(* IEC 61131-3 sources: FishAndCat/plc, 9 files *)

(* ---- 01_DUTs.st ---- *)
(* ============================================================
   01_DUTs.st — 数据类型定义(DUT)
   项目:智储优控 · 立体仓储仓位优化(2026 ABB杯 赛道一)
   目标平台:ABB AC500 V3(CODESYS V3.5 内核),ST 语言
   导入方法:Automation Builder 中 Application 右键 → 添加对象 → DUT,
            每个 TYPE 建一个 DUT,粘贴对应段落(详见 README_PLC.md)
   口径依据:docs/canonical_assumptions.md(A1-A9/B1-B5/C1-C8)
   ============================================================ *)

(* ---------- ST_Good:货物(题面五元组 + 分配结果字段) ---------- *)
TYPE ST_Good :
STRUCT
    Id          : INT;          // 序号(题面属性1)
    Name        : STRING[32];   // 名称(题面属性2)
    Weight      : REAL;         // 重量 kg(题面属性3)
    Freq        : REAL;         // 访问频次(题面属性4)
    Volume      : REAL;         // 体积 m3(题面属性5)
    Priority    : REAL;         // Rank阶段优先级(λ1*频次+λ2*重量+λ3*体积,归一后)
    Assigned    : BOOL;         // 是否已分配
    X           : INT;          // 分配结果:列(0..19,水平)
    Y           : INT;          // 分配结果:层(0..19,垂直,0=底层)
    Score       : REAL;         // 分配时的多目标评分
    PathLength  : REAL;         // 单程曼哈顿路径长度 m(口径C2)
    ExecTime    : REAL;         // 单程切比雪夫行程时间 s(口径C2)
END_STRUCT
END_TYPE

(* ---------- ST_Slot:仓位 ---------- *)
TYPE ST_Slot :
STRUCT
    X           : INT;          // 列 0..19
    Y           : INT;          // 层 0..19(0=底层)
    Occupied    : BOOL;         // 已占用(含预占用)
    PresetOcc   : BOOL;         // 预占用(题面:坐标能被3整除,解读见 FC_IsPresetOccupied)
    CapCoef     : REAL;         // 承重系数 = 1.0 - 0.02*Y(题面给定)
    MaxWeight   : REAL;         // 限重 = CapCoef * BASE_CAP(口径A6)
    MaxVolume   : REAL;         // 容积上限 = CELL_VOL(口径B4)
    GoodsId     : INT;          // 存放的货物Id,0=无
END_STRUCT
END_TYPE

(* ---------- ST_Stats:统计信息(决赛可视化统计栏数据源) ---------- *)
TYPE ST_Stats :
STRUCT
    PlacedCnt      : INT;       // 成功入库件数
    FailedCnt      : INT;       // 无可行位件数(边界:必须可见可报警)
    TotalTime2Way  : REAL;      // 入库总时间 s,双程口径(C1)
    AvgTime        : REAL;      // 平均单件双程时间 s
    ExpRetrieval   : REAL;      // 期望取货时间 s,频次加权单程(C3)
    Energy         : REAL;      // 能耗代理 Σ重量*高度 kg·m(C4)
    CogHeight      : REAL;      // 载荷重心高度 m(C6)
    PathTotal2Way  : REAL;      // 路径总长 m,双程曼哈顿(C5 损耗代理)
    UtilPct        : REAL;      // 空间利用率 =已占/400(C7,含预占)
    ViolCnt        : INT;       // 约束违规数,必须恒为0(C8)
    SwapCnt        : INT;       // 局部搜索接受的改进次数
    LsRounds       : INT;       // 局部搜索实际轮数
END_STRUCT
END_TYPE

(* ---------- E_MainState:主程序状态机 ---------- *)
TYPE E_MainState :
(
    STATE_IDLE       := 0,      // 待机
    STATE_INIT       := 10,     // 初始化仓库(预占用/承重)
    STATE_WAIT_INPUT := 20,     // 等待交互输入货物 / 载入演示批次
    STATE_ASSIGN     := 30,     // 批量分配运行中(分片,跨扫描周期)
    STATE_IMPROVE    := 40,     // 局部搜索改进中(分片,跨扫描周期)
    STATE_STATS      := 50,     // 统计计算
    STATE_DONE       := 60,     // 完成,结果可视化
    STATE_FAULT      := 70      // 故障(输入非法/无可行位等,看 GVL_Visu.StatusText)
);
END_TYPE

(* ---- 07_GVL_Data_generated.st ---- *)
(* ============================================================
   07_GVL_Data_generated.st — 生成文件,勿手改!
   由 sim/export_st_vectors.py 生成(seed=2026,N_DEMO=20,
   评分权重 α=1.0 β=0.6 γ=0.4 δ=0.15 = canonical E 默认)
   导入:TYPE 段建 DUT;GVL_Data 段建 GVL;FC_LoadDemoGoods 建 POU(函数)
   ============================================================ *)

(* ---------- DUT:ST_TestVec ---------- *)
TYPE ST_TestVec :
STRUCT
    W        : REAL;   // 货物重量
    F        : REAL;   // 货物频次
    X        : INT;    // 候选仓位列
    Y        : INT;    // 候选仓位层
    WMax     : REAL;   // 归一分母
    FMax     : REAL;
    ExpScore : REAL;   // Python 期望评分(双精度算出,容差1e-3比对)
    ExpTime  : REAL;   // Python 期望切比雪夫时间(匀速口径)
    ExpTimeAccel : REAL;   // Python 期望时间(L1 梯形加减速口径,T22 比对)
END_STRUCT
END_TYPE

(* ---------- DUT:ST_AwraCell(T25 终局布局向量) ---------- *)
TYPE ST_AwraCell :
STRUCT
    Id : INT;    // 货物序号
    X  : INT;    // 终局列
    Y  : INT;    // 终局层
END_STRUCT
END_TYPE

(* ---------- GVL:GVL_Data ---------- *)
VAR_GLOBAL CONSTANT
    N_DEMO    : INT := 20;
    N_TESTVEC : INT := 10;
    N_AWRA    : INT := 20;   // T25 终局向量件数
    AWRA_PLACED : INT := 20;
    AWRA_FAILED : INT := 0;
    LAM_F : REAL := 0.5;   // Rank λ 频次(单源,ST FC_CalcPriority 应引用)
    LAM_W : REAL := 0.35;   // Rank λ 重量
    LAM_V : REAL := 0.15;   // Rank λ 体积
    MAX_LS_ROUNDS : INT := 5;   // LS 最大轮数(单源,ST nMaxLsRounds 应引用)
END_VAR
VAR_GLOBAL
    aTestVec : ARRAY[1..10] OF ST_TestVec := [
        (W := 13.9, F := 1.83, X := 1, Y := 0, WMax := 80.0, FMax := 9.82, ExpScore := 0.122893, ExpTime := 0.500000, ExpTimeAccel := 2.828427),
        (W := 69.5, F := 1.1, X := 5, Y := 2, WMax := 80.0, FMax := 9.82, ExpScore := 0.222415, ExpTime := 4.000000, ExpTimeAccel := 6.324555),
        (W := 50.1, F := 2.02, X := 10, Y := 5, WMax := 80.0, FMax := 9.82, ExpScore := 0.306726, ExpTime := 10.000000, ExpTimeAccel := 11.666667),
        (W := 46.1, F := 3.1, X := 19, Y := 19, WMax := 80.0, FMax := 9.82, ExpScore := 0.891932, ExpTime := 38.000000, ExpTimeAccel := 39.666667),
        (W := 61.3, F := 2.14, X := 0, Y := 1, WMax := 80.0, FMax := 9.82, ExpScore := 0.162936, ExpTime := 2.000000, ExpTimeAccel := 3.666667),
        (W := 51.1, F := 1.11, X := 3, Y := 3, WMax := 80.0, FMax := 9.82, ExpScore := 0.230741, ExpTime := 6.000000, ExpTimeAccel := 7.666667),
        (W := 38.7, F := 4.28, X := 7, Y := 10, WMax := 80.0, FMax := 9.82, ExpScore := 0.524082, ExpTime := 20.000000, ExpTimeAccel := 21.666667),
        (W := 56.0, F := 1.23, X := 15, Y := 1, WMax := 80.0, FMax := 9.82, ExpScore := 0.166878, ExpTime := 7.500000, ExpTimeAccel := 11.500000),
        (W := 78.5, F := 9.82, X := 2, Y := 18, WMax := 80.0, FMax := 9.82, ExpScore := 1.876974, ExpTime := 36.000000, ExpTimeAccel := 37.666667),
        (W := 80.0, F := 1.86, X := 12, Y := 7, WMax := 80.0, FMax := 9.82, ExpScore := 0.514996, ExpTime := 14.000000, ExpTimeAccel := 15.666667)
    ];
    aAwraExpect : ARRAY[1..20] OF ST_AwraCell := [
        (Id := 1, X := 4, Y := 1),
        (Id := 2, X := 17, Y := 0),
        (Id := 3, X := 10, Y := 0),
        (Id := 4, X := 7, Y := 0),
        (Id := 5, X := 8, Y := 0),
        (Id := 6, X := 16, Y := 0),
        (Id := 7, X := 1, Y := 1),
        (Id := 8, X := 14, Y := 0),
        (Id := 9, X := 1, Y := 0),
        (Id := 10, X := 11, Y := 0),
        (Id := 11, X := 3, Y := 1),
        (Id := 12, X := 4, Y := 0),
        (Id := 13, X := 19, Y := 0),
        (Id := 14, X := 6, Y := 1),
        (Id := 15, X := 13, Y := 0),
        (Id := 16, X := 5, Y := 0),
        (Id := 17, X := 2, Y := 0),
        (Id := 18, X := 0, Y := 1),
        (Id := 19, X := 19, Y := 1),
        (Id := 20, X := 18, Y := 1)
    ];
    AWRA_EXPT   : REAL := 2.810626;   // 期望取货时间(ExpRetrieval 比对,容差1e-3)
    AWRA_ENERGY : REAL := 210.400000;  // 能耗 kg·m(Energy 比对)
    AWRA_COG    : REAL := 0.227632;     // 重心高(CogHeight 比对)
END_VAR

(* ---------- FC_LoadDemoGoods:载入演示批次(与 Python 仿真同源同 seed) ---------- *)
FUNCTION FC_LoadDemoGoods : BOOL
VAR
    n : INT;
END_VAR
n := GVL_WH.iGoodsCount;
n := n + 1;  GVL_WH.aGoods[n].Id := 1;  GVL_WH.aGoods[n].Name := 'G001';
GVL_WH.aGoods[n].Weight := 13.9;  GVL_WH.aGoods[n].Freq := 1.83;  GVL_WH.aGoods[n].Volume := 0.51;  GVL_WH.aGoods[n].Assigned := FALSE;
n := n + 1;  GVL_WH.aGoods[n].Id := 2;  GVL_WH.aGoods[n].Name := 'G002';
GVL_WH.aGoods[n].Weight := 69.5;  GVL_WH.aGoods[n].Freq := 1.1;  GVL_WH.aGoods[n].Volume := 0.28;  GVL_WH.aGoods[n].Assigned := FALSE;
n := n + 1;  GVL_WH.aGoods[n].Id := 3;  GVL_WH.aGoods[n].Name := 'G003';
GVL_WH.aGoods[n].Weight := 50.1;  GVL_WH.aGoods[n].Freq := 2.02;  GVL_WH.aGoods[n].Volume := 0.73;  GVL_WH.aGoods[n].Assigned := FALSE;
n := n + 1;  GVL_WH.aGoods[n].Id := 4;  GVL_WH.aGoods[n].Name := 'G004';
GVL_WH.aGoods[n].Weight := 46.1;  GVL_WH.aGoods[n].Freq := 3.1;  GVL_WH.aGoods[n].Volume := 0.71;  GVL_WH.aGoods[n].Assigned := FALSE;
n := n + 1;  GVL_WH.aGoods[n].Id := 5;  GVL_WH.aGoods[n].Name := 'G005';
GVL_WH.aGoods[n].Weight := 61.3;  GVL_WH.aGoods[n].Freq := 2.14;  GVL_WH.aGoods[n].Volume := 0.29;  GVL_WH.aGoods[n].Assigned := FALSE;
n := n + 1;  GVL_WH.aGoods[n].Id := 6;  GVL_WH.aGoods[n].Name := 'G006';
GVL_WH.aGoods[n].Weight := 51.1;  GVL_WH.aGoods[n].Freq := 1.11;  GVL_WH.aGoods[n].Volume := 0.75;  GVL_WH.aGoods[n].Assigned := FALSE;
n := n + 1;  GVL_WH.aGoods[n].Id := 7;  GVL_WH.aGoods[n].Name := 'G007';
GVL_WH.aGoods[n].Weight := 38.7;  GVL_WH.aGoods[n].Freq := 4.28;  GVL_WH.aGoods[n].Volume := 0.65;  GVL_WH.aGoods[n].Assigned := FALSE;
n := n + 1;  GVL_WH.aGoods[n].Id := 8;  GVL_WH.aGoods[n].Name := 'G008';
GVL_WH.aGoods[n].Weight := 56.0;  GVL_WH.aGoods[n].Freq := 1.23;  GVL_WH.aGoods[n].Volume := 0.3;  GVL_WH.aGoods[n].Assigned := FALSE;
n := n + 1;  GVL_WH.aGoods[n].Id := 9;  GVL_WH.aGoods[n].Name := 'G009';
GVL_WH.aGoods[n].Weight := 78.5;  GVL_WH.aGoods[n].Freq := 9.82;  GVL_WH.aGoods[n].Volume := 0.74;  GVL_WH.aGoods[n].Assigned := FALSE;
n := n + 1;  GVL_WH.aGoods[n].Id := 10;  GVL_WH.aGoods[n].Name := 'G010';
GVL_WH.aGoods[n].Weight := 80.0;  GVL_WH.aGoods[n].Freq := 1.86;  GVL_WH.aGoods[n].Volume := 0.16;  GVL_WH.aGoods[n].Assigned := FALSE;
n := n + 1;  GVL_WH.aGoods[n].Id := 11;  GVL_WH.aGoods[n].Name := 'G011';
GVL_WH.aGoods[n].Weight := 30.5;  GVL_WH.aGoods[n].Freq := 2.02;  GVL_WH.aGoods[n].Volume := 0.33;  GVL_WH.aGoods[n].Assigned := FALSE;
n := n + 1;  GVL_WH.aGoods[n].Id := 12;  GVL_WH.aGoods[n].Name := 'G012';
GVL_WH.aGoods[n].Weight := 39.3;  GVL_WH.aGoods[n].Freq := 6.07;  GVL_WH.aGoods[n].Volume := 0.66;  GVL_WH.aGoods[n].Assigned := FALSE;
n := n + 1;  GVL_WH.aGoods[n].Id := 13;  GVL_WH.aGoods[n].Name := 'G013';
GVL_WH.aGoods[n].Weight := 48.3;  GVL_WH.aGoods[n].Freq := 1.02;  GVL_WH.aGoods[n].Volume := 0.67;  GVL_WH.aGoods[n].Assigned := FALSE;
n := n + 1;  GVL_WH.aGoods[n].Id := 14;  GVL_WH.aGoods[n].Name := 'G014';
GVL_WH.aGoods[n].Weight := 32.3;  GVL_WH.aGoods[n].Freq := 1.6;  GVL_WH.aGoods[n].Volume := 0.42;  GVL_WH.aGoods[n].Assigned := FALSE;
n := n + 1;  GVL_WH.aGoods[n].Id := 15;  GVL_WH.aGoods[n].Name := 'G015';
GVL_WH.aGoods[n].Weight := 48.9;  GVL_WH.aGoods[n].Freq := 1.81;  GVL_WH.aGoods[n].Volume := 0.19;  GVL_WH.aGoods[n].Assigned := FALSE;
n := n + 1;  GVL_WH.aGoods[n].Id := 16;  GVL_WH.aGoods[n].Name := 'G016';
GVL_WH.aGoods[n].Weight := 43.0;  GVL_WH.aGoods[n].Freq := 3.31;  GVL_WH.aGoods[n].Volume := 0.58;  GVL_WH.aGoods[n].Assigned := FALSE;
n := n + 1;  GVL_WH.aGoods[n].Id := 17;  GVL_WH.aGoods[n].Name := 'G017';
GVL_WH.aGoods[n].Weight := 41.8;  GVL_WH.aGoods[n].Freq := 8.53;  GVL_WH.aGoods[n].Volume := 0.31;  GVL_WH.aGoods[n].Assigned := FALSE;
n := n + 1;  GVL_WH.aGoods[n].Id := 18;  GVL_WH.aGoods[n].Name := 'G018';
GVL_WH.aGoods[n].Weight := 36.5;  GVL_WH.aGoods[n].Freq := 9.46;  GVL_WH.aGoods[n].Volume := 0.48;  GVL_WH.aGoods[n].Assigned := FALSE;
n := n + 1;  GVL_WH.aGoods[n].Id := 19;  GVL_WH.aGoods[n].Name := 'G019';
GVL_WH.aGoods[n].Weight := 43.8;  GVL_WH.aGoods[n].Freq := 1.02;  GVL_WH.aGoods[n].Volume := 0.28;  GVL_WH.aGoods[n].Assigned := FALSE;
n := n + 1;  GVL_WH.aGoods[n].Id := 20;  GVL_WH.aGoods[n].Name := 'G020';
GVL_WH.aGoods[n].Weight := 14.7;  GVL_WH.aGoods[n].Freq := 1.04;  GVL_WH.aGoods[n].Volume := 0.66;  GVL_WH.aGoods[n].Assigned := FALSE;
GVL_WH.iGoodsCount := n;
FC_LoadDemoGoods := TRUE;
END_FUNCTION

(* ---- 02_GVL.st ---- *)
(* ============================================================
   02_GVL.st — 全局变量列表
   导入方法:Application 右键 → 添加对象 → 全局变量列表(GVL),
            建三个 GVL:GVL_Param / GVL_WH / GVL_Visu,分别粘贴对应段落
   注意:参数与 Python 仿真 sim/warehouse_sim.py 顶部常量一一对应,
        改任何一边必须同步另一边并重跑一致性向量(README_PLC.md 流程)
   ============================================================ *)

(* ---------- GVL_Param:场景与算法参数 ---------- *)
VAR_GLOBAL CONSTANT
    COLS        : INT  := 20;       // 列数(A1)
    TIERS       : INT  := 20;       // 层数(A1)
    MAX_GOODS   : INT  := 400;      // 货物数组上限(=仓位总数)
    CELL_W      : REAL := 1.0;      // 仓位宽 m(A2)
    CELL_H      : REAL := 1.0;      // 仓位高 m(A2)
    BASE_CAP    : REAL := 100.0;    // 底层限重 kg(A6)
    CELL_VOL    : REAL := 1.0;      // 仓位容积 m3(B4)
    // ---- L6 可视化画面几何常量(单位 px;与 2_你要操作/AB可视化搭建操作卡 的元件坐标同源) ----
    GRID_X0     : INT := 40;        // 仓位网格左上角 X(左侧留层号标签)
    GRID_Y0     : INT := 40;        // 仓位网格左上角 Y(顶部留标题)
    CELL_PX_W   : INT := 28;        // 单格宽(20列=560px,网格右缘 x=600)
    CELL_PX_H   : INT := 20;        // 单格高(20层=400px,网格下缘 y=440)
    // ---- A4 两级权限(0711):演示 PIN,非真实凭据;变量层方案依据=内置 visu
    //      Access Rights 无 ScriptEngine 接口,无法被画面生成管线驱动(官方文档核实) ----
    ADMIN_PIN   : INT := 2026;      // 管理员登录码(演示口径;生产化换 visu UserMgmt)
END_VAR

VAR_GLOBAL
    // ---- 设备参数(A4;非常量:答辩时可现场演示灵敏度) ----
    rVx             : REAL := 2.0;      // 堆垛机水平速度 m/s
    rVy             : REAL := 0.5;      // 堆垛机垂直速度 m/s
    rTLoad          : REAL := 0.0;      // 装货时间 s(A8:暂不计,保留接口)
    rTUnload        : REAL := 0.0;      // 卸货时间 s(A8)
    xSimultaneousXY : BOOL := TRUE;     // TRUE=切比雪夫(主口径A5) FALSE=顺序模型(A9对照)
    // ---- L1 梯形速度曲线(A4b;与 Python ACCEL/AX/AY 一字对齐) ----
    xUseAccel       : BOOL := FALSE;    // FALSE=匀速(基础口径,历史数字) TRUE=加减速工程口径
    rAx             : REAL := 0.5;      // 水平加减速 m/s²
    rAy             : REAL := 0.3;      // 垂直加减速 m/s²

    // ---- U2 载重运动学(块3 拟真调参区,画面可调;默认=canonical U2/sim 同值) ----
    // 消费者:FC_TravelLaden(垂直折减)/FC_HandleTime(装卸三档);不进现有评分/测试链路(零回归)
    rLadenFactorVY  : REAL := 0.80;     // 满载垂直速度折减(Mecalux 0.818 圆整,水平不折减=行业惯例)
    rHandleW1       : REAL := 30.0;     // 装卸档界1:轻货上限 kg
    rHandleW2       : REAL := 60.0;     // 装卸档界2:中货上限 kg(>W2 为重货)
    rHandleT1       : REAL := 6.0;      // 轻货装卸 s(单次货叉全循环)
    rHandleT2       : REAL := 8.5;      // 中货装卸 s
    rHandleT3       : REAL := 12.5;     // 重货装卸 s

    // ---- 预占用规则(B1;2026-07-06 官方答复后默认=3,四解读全保留可切) ----
    iPreRule        : INT := 3;         // 3=x+y被3整除(133格,官方口径) 0=且(49格) 1=或(231格) 2=线性(134格)

    // ---- 多目标评分权重(canonical E,HMI 可调,默认=Python 标定值) ----
    rAlpha          : REAL := 1.0;      // 效率项:频次*时间
    rBeta           : REAL := 0.6;      // 稳定项:重量*层高
    rGamma          : REAL := 0.4;      // 能耗项:提升做功
    rDelta          : REAL := 0.15;     // 位置价值预留项(δ=0会退化成就近贪心,实验发现F2)

    // ---- AWRA-LS Rank 权重(canonical E) ----
    rLambda1        : REAL := 0.50;     // 频次优先
    rLambda2        : REAL := 0.35;     // 重量优先(紧库存下保证重货有低层位,实验发现F3)
    rLambda3        : REAL := 0.15;     // 体积优先

    // ---- 扫描周期分片参数(非阻塞设计:单周期计算量受控,防看门狗超时) ----
    nBatchPerCycle  : INT := 10;        // 分配阶段:每扫描周期处理货物件数
    nPairsPerCycle  : INT := 200;       // 局部搜索:每扫描周期评估交换对数
    nMaxLsRounds    : INT := 5;         // 局部搜索最大轮数(120件实测2-3轮收敛)
END_VAR

(* ---------- GVL_WH:仓库与货物运行数据 ---------- *)
VAR_GLOBAL
    aSlots      : ARRAY[0..19, 0..19] OF ST_Slot;   // [列,层]
    aGoods      : ARRAY[1..400] OF ST_Good;          // 货物表(1..iGoodsCount 有效)
    iGoodsCount : INT := 0;                          // 当前货物数
    aRankIdx    : ARRAY[1..400] OF INT;              // Rank阶段排序后的货物下标
    stStats     : ST_Stats;                          // 统计结果
    // ---- A3 检修挂起(0711):独立于 aSlots 的物理状态层,Reset/重分配不清
    //      语义=SAP EWM bin blocking 的 putaway block:禁新入库(选位/分配/交换均排除),
    //      已有货物原地冻结、查询照常;非 RETAIN(断电清零=演示安全默认) ----
    aMaintBlock : ARRAY[0..19, 0..19] OF BOOL;       // TRUE=该格检修挂起
    // ---- C2/C6 热力图数据层(0711 批次前置令) ----
    aSlotFreq   : ARRAY[0..19, 0..19] OF REAL;       // C2:格上货物频次(布局态,fbInit 清)
    aSlotOps    : ARRAY[0..19, 0..19] OF INT;        // C6:存取履历计数(放置/搬移/交换各+1;
                                                     //     物理履历,Reset 不清,同 aMaintBlock 语义)
END_VAR

(* ---------- GVL_Visu:可视化接口(决赛 CODESYS Visualization 绑定这里) ----------
   资料包 §10.2 结构,状态编码:
   0=空闲(浅灰) 1=预占用(深灰) 2=已占用(绿) 3=当前推荐(黄) 4=路径(蓝) 5=报警(红) *)
VAR_GLOBAL
    VisuSlotState   : ARRAY[0..19, 0..19] OF INT;
    VisuCurrentX    : INT;                  // 堆垛机当前位置(演示动画用)
    VisuCurrentY    : INT;
    VisuTargetX     : INT;                  // 当前目标仓位
    VisuTargetY     : INT;
    VisuPathX       : ARRAY[0..39] OF INT;  // 当前路径点序列(L形:先水平后垂直展开)
    VisuPathY       : ARRAY[0..39] OF INT;
    VisuPathCount   : INT;
    VisuPathLen     : REAL;                 // 当前路径长度 m(曼哈顿,口径C2)
    VisuExecTime    : REAL;                 // 当前执行时间 s(切比雪夫,口径C2)
    VisuStatusText  : STRING[128];          // 状态/报警文本
    // ---- 统计面板(FB_Stats 写入) ----
    VisuTotalTime          : REAL;          // 完成全部存储总时间 s(双程,C1)
    VisuAvgTime            : REAL;          // 平均单件时间 s
    VisuSpaceUtilization   : REAL;          // 空间利用率(C7)
    VisuWearIndex          : REAL;          // 设备损耗代理=路径总长 m(C5)
    VisuViolationCount     : INT;           // 违规数(C8,恒0)
    // ---- 输入区(HMI 交互:决赛"可通过交互界面输入货物属性"要求) ----
    InGoodId        : INT;
    InGoodName      : STRING[32];
    InGoodWeight    : REAL;
    InGoodFreq      : REAL;
    InGoodVolume    : REAL;
    CmdAddGood      : BOOL;                 // 按钮:添加单件货物
    CmdLoadDemo     : BOOL;                 // 按钮:载入演示批次(Python seed=2026 导出)
    CmdRunAssign    : BOOL;                 // 按钮:运行批量分配(AWRA-LS)
    CmdReset        : BOOL;                 // 按钮:复位重来
    SelStrategy     : INT := 2;             // 策略选择 0=seq 1=near 2=score(在线) 3=AWRA-LS(批量)
    // ---- L6 决赛画面增补(元件绑定方法见 2_你要操作/AB可视化搭建操作卡.md) ----
    VisuSlotColor   : ARRAY[0..19, 0..19] OF DWORD;
        // [列,显示行] 单元格填充色(16#00RRGGBB);显示行0=画面顶(=层19),
        // 上下翻转+状态→颜色查表由 FB_VisuRefresh 每周期重算——画面矩形阵列只绑这一个数组
    VisuCraneXpx    : INT;                  // 堆垛机图元 X 像素(FB_VisuRefresh 从 VisuCurrentX 换算)
    VisuCraneYpx    : INT;                  // 堆垛机图元 Y 像素(含上下翻转)
    VisuAlarm       : BOOL;                 // 报警灯:超重/负输入/无可行位=TRUE(演示第6步,红灯元件)
    CmdAnimate      : BOOL;                 // 按钮:堆垛机沿当前路径回放动画(FB_AnimatePath)
    // ---- 块3 P3 单件查询页(评分细则8"单件查询";FB_QueryGood 填充,状态6=青色高亮) ----
    InQueryId       : INT;                  // 查询输入:货物序号
    CmdQuery        : BOOL;                 // 按钮:执行查询
    QryFound        : BOOL;                 // 查到与否(FALSE 时下方字段无效)
    QryX            : INT;                  // 位置列
    QryY            : INT;                  // 位置层
    QryName         : STRING[32];
    QryWeight       : REAL;
    QryFreq         : REAL;
    QryVolume       : REAL;
    QryPathLen      : REAL;                 // 路径长度 m(曼哈顿,C2)
    QryExecTime     : REAL;                 // 行程时间 s(切比雪夫单程,存量口径)
    QryTravelLaden  : REAL;                 // 载货行程 s(垂直×rLadenFactorVY,U2 拟真对照)
    QryHandleT      : REAL;                 // 单次装卸 s(三档,U2)——调参区改档界/时长此值实时变
    // ---- 块3 P2 统计记录页(评分细则8;FB_RecordPage 10 行窗口映射,禁 400 行整表压渲染) ----
    iRecTop         : INT;                  // 窗口顶行(1 基,指向 aGoods 下标)
    CmdPageUp       : BOOL;                 // 按钮:上翻 10 行
    CmdPageDown     : BOOL;                 // 按钮:下翻 10 行
    iRecTotal       : INT;                  // 总行数(=iGoodsCount,表头"共 N 件"用)
    aRowId          : ARRAY[0..9] OF INT;   // 10 行窗口:序号(0=空行)
    aRowX           : ARRAY[0..9] OF INT;   // 位置列(未分配=-1)
    aRowY           : ARRAY[0..9] OF INT;   // 位置层
    aRowPathLen     : ARRAY[0..9] OF REAL;  // 路径长度 m
    aRowExecT       : ARRAY[0..9] OF REAL;  // 行程时间 s
    // ---- 块3 快照对比(方向9:一键切换"优化前 vs 优化后",D 档叙事) ----
    CmdSaveSnap     : BOOL;                 // 按钮:把当前布局存为对比基准(如 seq 基线)
    CmdCompareMode  : BOOL;                 // 开关:TRUE=显示快照 FALSE=显示实时(FB_VisuRefresh 选源)
    xSnapValid      : BOOL;                 // 已存过快照(未存时 CompareMode 无效,防显示垃圾)
    aSnapState      : ARRAY[0..19, 0..19] OF INT;  // 快照:VisuSlotState 的冻结副本
    // ---- 块3 名称下拉+手输(ComboBox Array 写 INT 下标,PRG 同步回 InGoodName) ----
    iNameSel        : INT := -1;            // ComboBox 选中下标(-1=未选,手输优先)
    astrNames       : ARRAY[0..9] OF STRING[32] :=
        ['BEARING','MOTOR','GEARBOX','VALVE','PUMP','SENSOR','CABLE','PANEL','FILTER','RELAY'];
        // 常用货物名(ASCII,C0555 规避;演示可选,亦可 Keypad 手输)
    // ---- 块3 画面排版 B(0710):装饰/图例常量——脚本设不了静态填色(0710 实证),
    //      全部走已验证的 Color variables 动态通道;RGBA 前导 FF=不透明,00=全透明 ----
    dwCraneColor    : DWORD := 16#FFFF6D00;         // 堆垛机橙
    dwTransparent   : DWORD := 16#00FFFFFF;         // 全透明填充(分组框矩形只显边线,不盖内容)
    dwHeaderBg      : DWORD := 16#FFE8EAF0;         // P2 记录表表头底纹(版1 排版,0711)
    aLegendColor    : ARRAY[0..7] OF DWORD :=       // 图例色样,与 FC_StateToColor 状态 0..7 一致
        [16#FFE8E8E8, 16#FF707070, 16#FF43A047, 16#FFFFC107,
         16#FF42A5F5, 16#FFE53935, 16#FF26C6DA, 16#FF8E24AA];
    // ---- A2 场景检测器(0711 驾驶舱连击:批次画像→推荐策略;FB_SceneDetect 填充) ----
    VisuProfN       : INT;                  // 画像:批量大小
    VisuProfDensity : REAL;                 // 画像:密度 n/267(sum 口径可用位)
    VisuProfSkew    : REAL;                 // 画像:频次偏斜度(top20% 件频次占比)
    VisuProfWMean   : REAL;                 // 画像:重量均值 kg
    VisuProfWHeavy  : REAL;                 // 画像:重货(>60kg)占比
    VisuRecStrategy : INT := -1;            // 推荐策略档位(SelStrategy 语义;-1=无数据)
    VisuRecText     : STRING[64];           // 推荐文本(ASCII 状态码,画面静态中文标签对照)
    xAutoStrategy   : BOOL := FALSE;        // 开关:TRUE=推荐自动写入 SelStrategy(人工覆盖=关)
    // ---- A3 检修画面接口 ----
    InMaintX        : INT;                  // 检修目标列
    InMaintY        : INT;                  // 检修目标层
    CmdMaintToggle  : BOOL;                 // 按钮:挂起/恢复翻转(需管理员)
    VisuMaintCount  : INT;                  // 当前检修格数
    // ---- C1/C2/C6 视图层(0711 批次前置令:层高亮+双热力图,画面终局一次施工) ----
    iViewMode       : INT := 0;             // 0=状态视图 1=频次热力(C2) 2=损耗热力(C6)
    CmdViewCycle    : BOOL;                 // 按钮:视图循环切换(脉冲)
    InTierSel       : INT := -1;            // C1 层高亮选择(-1=关,0..19=该层加亮)
    VisuTierOcc     : INT;                  // C1:选中层的在货格数(FB_VisuRefresh 计)
    // ---- A4 两级权限画面接口(变量层双闸:画面元素锁定 + ST 侧参数守卫回滚) ----
    InPinCode       : INT;                  // 登录码输入(消费即清,画面不放回显元件)
    CmdLogin        : BOOL;                 // 按钮:登录
    CmdLogout       : BOOL;                 // 按钮:登出
    iUserLevel      : INT := 0;             // 0=操作员 1=管理员(画面锁定绑定源;非 RETAIN)
    VisuUserText    : STRING[32];           // 'USER=OPERATOR' / 'USER=ADMIN' / 'LOGIN_FAIL'
END_VAR

(* ---- 08_GVL_WeightPolicy_generated.st ---- *)
(* ============================================================
   08_GVL_WeightPolicy_generated.st — 生成文件,勿手改!
   由 sim/adaptive_weights.py 生成:场景→权重 策略表(A1 自适应机制)
   场景判档(PLC 在线可算):iDensity 0/1/2=占用率<55%/<85%/其余;
   iDist 0/1/2=均匀/高频偏态/重货(按库存重量均值与频次变异系数判,见 FC_ClassifyScene);
   xBatch FALSE=在线逐件 TRUE=批量重排。
   ============================================================ *)
VAR_GLOBAL CONSTANT
    // aPolicyDelta/aPolicyBG[iDensity, iDist, xBatch(0/1)]
    aPolicyDelta : ARRAY[0..2, 0..2, 0..1] OF REAL := [
        0.2, 0.15, 0.1, 0.05, 0.1, 0.1, 0.2, 0.15, 0.2, 0.05, 0.2, 0.15, 0.2, 0.2, 0.2, 0.05, 0.2, 0.2];
    aPolicyBG : ARRAY[0..2, 0..2, 0..1] OF REAL := [
        0.6, 0.6, 1.0, 0.6, 0.6, 0.6, 0.6, 0.6, 0.6, 0.6, 0.6, 0.6, 0.6, 0.6, 0.6, 0.6, 0.6, 0.6];
END_VAR

(* 用法(PRG_Main 分配启动前调用):
   GVL_Param.rDelta := aPolicyDelta[iDensity, iDist, SEL(xBatch, 0, 1)];
   bg := aPolicyBG[iDensity, iDist, SEL(xBatch, 0, 1)];
   GVL_Param.rBeta := bg / 2.0;  GVL_Param.rGamma := bg / 2.0;  *)

(* ---- 03_Functions.st ---- *)
(* ============================================================
   03_Functions.st — 纯函数(FC,无状态,可单元测试)
   导入方法:Application 右键 → 添加对象 → POU,类型选"功能(Function)",
            每个 FUNCTION 建一个 POU,粘贴对应段落
   一致性:每个函数与 sim/warehouse_sim.py 同名逻辑一字对齐,
          由 sim/export_st_vectors.py 生成的测试向量在 PRG_Test 中比对
   ============================================================ *)

(* ---------- FC_CapCoef:层承重系数(题面:底层1.0,每层-0.02) ---------- *)
FUNCTION FC_CapCoef : REAL
VAR_INPUT
    y : INT;                    // 层号 0..19
END_VAR
VAR
    yy : INT;
END_VAR
// 边界:越界钳位(边界判断清单#1)
IF y < 0 THEN
    yy := 0;
ELSIF y > GVL_Param.TIERS - 1 THEN
    yy := GVL_Param.TIERS - 1;
ELSE
    yy := y;
END_IF
FC_CapCoef := 1.0 - 0.02 * INT_TO_REAL(yy);
END_FUNCTION

(* ---------- FC_IsPresetOccupied:预占用判定(B1 四解读封装;官方口径=3,2026-07-06 答复落地) ---------- *)
FUNCTION FC_IsPresetOccupied : BOOL
VAR_INPUT
    x     : INT;
    y     : INT;
    iRule : INT;                // 3=sum(133格,官方) 0=and(49格) 1=or(231格) 2=linear(134格)
END_VAR
FC_IsPresetOccupied := FALSE;
IF x < 0 OR x > GVL_Param.COLS - 1 OR y < 0 OR y > GVL_Param.TIERS - 1 THEN
    RETURN;                     // 越界视为不可用由 FC_CheckFeasible 把关,这里仅答"是否预占"
END_IF
CASE iRule OF
    3: FC_IsPresetOccupied := ((x + y) MOD 3 = 0);            // 官方口径(0706):x+y 之和能被3整除
    0: FC_IsPresetOccupied := (x MOD 3 = 0) AND (y MOD 3 = 0);
    1: FC_IsPresetOccupied := (x MOD 3 = 0) OR  (y MOD 3 = 0);
    2: FC_IsPresetOccupied := ((x * GVL_Param.TIERS + y) MOD 3 = 0);
ELSE
    FC_IsPresetOccupied := ((x + y) MOD 3 = 0);               // 非法规则回落官方口径
END_CASE
END_FUNCTION

(* ---------- FC_CheckFeasible:仓位可行性(边界判断核心) ---------- *)
FUNCTION FC_CheckFeasible : BOOL
VAR_INPUT
    x          : INT;           // 目标仓位
    y          : INT;
    rGoodW     : REAL;          // 货物重量
    rGoodV     : REAL;          // 货物体积
END_VAR
FC_CheckFeasible := FALSE;
// 边界清单:越界 / 负属性 / 检修挂起 / 占用(含预占) / 超重 / 超容积
IF x < 0 OR x > GVL_Param.COLS - 1 OR y < 0 OR y > GVL_Param.TIERS - 1 THEN RETURN; END_IF
IF rGoodW < 0.0 OR rGoodV < 0.0 THEN RETURN; END_IF
IF GVL_WH.aMaintBlock[x, y] THEN RETURN; END_IF      // A3 putaway block:检修位禁新入库
IF GVL_WH.aSlots[x, y].Occupied THEN RETURN; END_IF
IF rGoodW > GVL_WH.aSlots[x, y].MaxWeight THEN RETURN; END_IF
IF rGoodV > GVL_WH.aSlots[x, y].MaxVolume THEN RETURN; END_IF
FC_CheckFeasible := TRUE;
END_FUNCTION

(* ---------- FC_FitsPhysical:仅物理约束(局部交换用:目标位即将腾出,不查占用) ---------- *)
FUNCTION FC_FitsPhysical : BOOL
VAR_INPUT
    x      : INT;
    y      : INT;
    rGoodW : REAL;
    rGoodV : REAL;
END_VAR
FC_FitsPhysical := FALSE;
IF x < 0 OR x > GVL_Param.COLS - 1 OR y < 0 OR y > GVL_Param.TIERS - 1 THEN RETURN; END_IF
IF rGoodW < 0.0 OR rGoodV < 0.0 THEN RETURN; END_IF
// A3:交换目标位检修中=禁入(检修位上的货可被换走,但别的货不得换进来——
//     与 SAP EWM putaway block"存量可出、新增禁入"语义一致)
IF GVL_WH.aMaintBlock[x, y] THEN RETURN; END_IF
IF rGoodW > GVL_WH.aSlots[x, y].MaxWeight THEN RETURN; END_IF
IF rGoodV > GVL_WH.aSlots[x, y].MaxVolume THEN RETURN; END_IF
FC_FitsPhysical := TRUE;
END_FUNCTION

(* ---------- FC_AxisTime:L1 单轴行程时间(梯形/三角速度曲线) ----------
   与 Python axis_time 一字对齐:d≥v²/a → d/v+v/a(梯形);否则 2·√(d/a)(三角)。
   匀速模型系统性低估短程时间(实验发现 F7:对优化布局低估 43.5%)。 *)
FUNCTION FC_AxisTime : REAL
VAR_INPUT
    d    : REAL;                // 行程距离 m(非负)
    vmax : REAL;                // 峰值速度 m/s
    acc  : REAL;                // 加减速 m/s²
END_VAR
IF d <= 0.0 THEN
    FC_AxisTime := 0.0;
    RETURN;
END_IF
IF vmax <= 0.0 THEN vmax := 1.0; END_IF     // 非法输入保护
IF acc  <= 0.0 THEN acc  := 0.1; END_IF
IF d >= vmax * vmax / acc THEN
    FC_AxisTime := d / vmax + vmax / acc;
ELSE
    FC_AxisTime := 2.0 * SQRT(d / acc);
END_IF
END_FUNCTION

(* ---------- FC_CalcTravelTime:行程时间(A5/A9/A4b 三开关) ----------
   主口径 = 切比雪夫:双电机同动取慢轴;xSimXY=FALSE 退化为顺序模型(对照)。
   GVL_Param.xUseAccel=TRUE 时轴时间用梯形曲线(L1 工程口径),与 Python 同全局开关。 *)
FUNCTION FC_CalcTravelTime : REAL
VAR_INPUT
    x0, y0, x1, y1  : INT;      // 起点/终点(格坐标;支持任意两点,双命令周期用)
    xSimXY          : BOOL;     // TRUE=切比雪夫 FALSE=顺序
END_VAR
VAR
    dx, dy, tx, ty : REAL;
    vx, vy         : REAL;
END_VAR
dx := ABS(INT_TO_REAL(x1 - x0)) * GVL_Param.CELL_W;
dy := ABS(INT_TO_REAL(y1 - y0)) * GVL_Param.CELL_H;
// 边界:速度非法保护(边界清单#8思想:非法输入修正)
vx := GVL_Param.rVx;  IF vx <= 0.0 THEN vx := 1.0; END_IF
vy := GVL_Param.rVy;  IF vy <= 0.0 THEN vy := 1.0; END_IF
IF GVL_Param.xUseAccel THEN
    tx := FC_AxisTime(d := dx, vmax := vx, acc := GVL_Param.rAx);
    ty := FC_AxisTime(d := dy, vmax := vy, acc := GVL_Param.rAy);
ELSE
    tx := dx / vx;
    ty := dy / vy;
END_IF
IF xSimXY THEN
    FC_CalcTravelTime := MAX(tx, ty) + GVL_Param.rTLoad + GVL_Param.rTUnload;
ELSE
    FC_CalcTravelTime := tx + ty + GVL_Param.rTLoad + GVL_Param.rTUnload;
END_IF
END_FUNCTION

(* ---------- FC_CalcDualCycleTime:L2 双命令周期时间(C10 口径) ----------
   一趟联合行程:I/O→存位(带货)→取位(空驶联程)→I/O(带货);
   节省 = 单命令(2t存+2t取) − 本值 ≥ 0(切比雪夫三角不等式,有 Python 测试)。 *)
FUNCTION FC_CalcDualCycleTime : REAL
VAR_INPUT
    iStoreX, iStoreY : INT;     // 存位
    iRetrX,  iRetrY  : INT;     // 取位
END_VAR
FC_CalcDualCycleTime :=
      FC_CalcTravelTime(x0 := 0, y0 := 0, x1 := iStoreX, y1 := iStoreY,
                        xSimXY := GVL_Param.xSimultaneousXY)
    + FC_CalcTravelTime(x0 := iStoreX, y0 := iStoreY, x1 := iRetrX, y1 := iRetrY,
                        xSimXY := GVL_Param.xSimultaneousXY)
    + FC_CalcTravelTime(x0 := iRetrX, y0 := iRetrY, x1 := 0, y1 := 0,
                        xSimXY := GVL_Param.xSimultaneousXY);
END_FUNCTION

(* ---------- FC_CalcPathLen:路径长度(曼哈顿,口径C2:与时间并列呈现不混用) ---------- *)
FUNCTION FC_CalcPathLen : REAL
VAR_INPUT
    x0, y0, x1, y1 : INT;
END_VAR
FC_CalcPathLen := ABS(INT_TO_REAL(x1 - x0)) * GVL_Param.CELL_W
                + ABS(INT_TO_REAL(y1 - y0)) * GVL_Param.CELL_H;
END_FUNCTION

(* ---------- FC_TMax:全库最远仓位单程时间(评分归一分母) ---------- *)
FUNCTION FC_TMax : REAL
FC_TMax := MAX(INT_TO_REAL(GVL_Param.COLS - 1) * GVL_Param.CELL_W / GVL_Param.rVx,
               INT_TO_REAL(GVL_Param.TIERS - 1) * GVL_Param.CELL_H / GVL_Param.rVy);
END_FUNCTION

(* ---------- FC_CalcScore:多目标评分(与 Python make_score_fn 一字对齐) ----------
   score = α·(频次/最大)·(时间/最大)   效率:高频货放远处要罚
         + β·(重量/最大)·(层/最高层)   稳定:重货放高层要罚
         + γ·(重量·高度)/(最大做功)    能耗:提升做功要罚(绿色指标)
         + δ·(1-频次归一)·(1-时间归一) 预留:冷门货占近位要罚(F2:无此项退化为就近贪心)
   注意:时间项用切比雪夫(xSimultaneousXY=TRUE 的主口径),归一分母 FC_TMax  *)
FUNCTION FC_CalcScore : REAL
VAR_INPUT
    rGoodW  : REAL;             // 货物重量
    rGoodF  : REAL;             // 货物频次
    x, y    : INT;              // 候选仓位
    rWMax   : REAL;             // 当前批次最大重量(归一)
    rFMax   : REAL;             // 当前批次最大频次(归一)
END_VAR
VAR
    tNorm, fNorm, hMax : REAL;
    eff, stab, energy, resv : REAL;
END_VAR
// 边界:归一分母保护
IF rWMax <= 0.0 THEN rWMax := 1.0; END_IF
IF rFMax <= 0.0 THEN rFMax := 1.0; END_IF
hMax := INT_TO_REAL(GVL_Param.TIERS - 1) * GVL_Param.CELL_H;

tNorm  := FC_CalcTravelTime(x0 := 0, y0 := 0, x1 := x, y1 := y,
                            xSimXY := GVL_Param.xSimultaneousXY) / FC_TMax();
fNorm  := rGoodF / rFMax;
eff    := fNorm * tNorm;
stab   := (rGoodW / rWMax) * (INT_TO_REAL(y) / INT_TO_REAL(GVL_Param.TIERS - 1));
energy := (rGoodW * INT_TO_REAL(y) * GVL_Param.CELL_H) / (rWMax * hMax);
resv   := (1.0 - fNorm) * (1.0 - tNorm);

FC_CalcScore := GVL_Param.rAlpha * eff + GVL_Param.rBeta * stab
              + GVL_Param.rGamma * energy + GVL_Param.rDelta * resv;
END_FUNCTION

(* ---------- FC_CalcPriority:Rank 阶段优先级(AWRA-LS 第一段) ----------
   高频、重、大体积优先分配 —— λ2 重量权重保证紧库存下重货先占低层(F3) *)
FUNCTION FC_CalcPriority : REAL
VAR_INPUT
    rGoodF : REAL;
    rGoodW : REAL;
    rGoodV : REAL;
    rFMax  : REAL;
    rWMax  : REAL;
    rVMax  : REAL;
END_VAR
IF rFMax <= 0.0 THEN rFMax := 1.0; END_IF
IF rWMax <= 0.0 THEN rWMax := 1.0; END_IF
IF rVMax <= 0.0 THEN rVMax := 1.0; END_IF
FC_CalcPriority := GVL_Param.rLambda1 * rGoodF / rFMax
                 + GVL_Param.rLambda2 * rGoodW / rWMax
                 + GVL_Param.rLambda3 * rGoodV / rVMax;
END_FUNCTION

(* ---------- FC_StateToColor:仓位状态码 → 画面填充色(L6 可视化) ----------
   颜色 DWORD 格式 = RGBA 16#AARRGGBB,前导字节 AA 为透明度:FF=不透明,00=全透明
   (官方 "Color definition in RGBA color space";AB2.9 Visualization Manager 的
   半透明绘制默认开启,前导字节按 alpha 解释——0710 实证:16#00RRGGBB 渲染为全透明,
   画面 400 格因此"看不见颜色",修为 16#FF 前缀)。
   状态编码与 GVL_Visu.VisuSlotState 注释一一对应:0空闲/1预占/2占用/3推荐/4路径/5报警。
   改配色只改这里——画面 400 个矩形元件不写死任何颜色(单一真相源)。 *)
FUNCTION FC_StateToColor : DWORD
VAR_INPUT
    iState : INT;
END_VAR
CASE iState OF
    0: FC_StateToColor := 16#FFE8E8E8;   // 空闲:浅灰
    1: FC_StateToColor := 16#FF707070;   // 预占用:深灰
    2: FC_StateToColor := 16#FF43A047;   // 已占用:绿
    3: FC_StateToColor := 16#FFFFC107;   // 当前推荐:黄
    4: FC_StateToColor := 16#FF42A5F5;   // 路径:蓝
    5: FC_StateToColor := 16#FFE53935;   // 报警:红
    6: FC_StateToColor := 16#FF26C6DA;   // 查询高亮:青(块3 P3,FB_QueryGood 置位)
    7: FC_StateToColor := 16#FF8E24AA;   // 检修挂起:紫(A3,FB_VisuRefresh 按 aMaintBlock 叠加)
ELSE
    FC_StateToColor := 16#FFFF00FF;      // 未知状态:品红(醒目,便于发现bug)
END_CASE
END_FUNCTION

(* ---------- FC_MaintToggle:检修挂起/恢复翻转(A3,0711) ----------
   语义=SAP EWM bin blocking 的 putaway block:挂起只禁"新入库"(FC_CheckFeasible/
   FC_FitsPhysical 已排除),已有货物原地冻结、查询照常;恢复即重新入分配池。
   需管理员(iLevel>=1)——检修是设备物理操作,权限门与 A4 联动。
   返回码:0=已挂起 1=已恢复 2=需管理员 3=坐标越界。
   带副作用(写 GVL_WH.aMaintBlock / GVL_Visu.VisuMaintCount),风格同 FC_LoadDemoGoods。 *)
FUNCTION FC_MaintToggle : INT
VAR_INPUT
    x      : INT;
    y      : INT;
    iLevel : INT;               // 当前用户级(FB_UserAuth 输出)
END_VAR
IF iLevel < 1 THEN
    FC_MaintToggle := 2;  RETURN;
END_IF
IF x < 0 OR x > GVL_Param.COLS - 1 OR y < 0 OR y > GVL_Param.TIERS - 1 THEN
    FC_MaintToggle := 3;  RETURN;
END_IF
IF GVL_WH.aMaintBlock[x, y] THEN
    GVL_WH.aMaintBlock[x, y] := FALSE;
    GVL_Visu.VisuMaintCount := GVL_Visu.VisuMaintCount - 1;
    FC_MaintToggle := 1;
ELSE
    GVL_WH.aMaintBlock[x, y] := TRUE;
    GVL_Visu.VisuMaintCount := GVL_Visu.VisuMaintCount + 1;
    FC_MaintToggle := 0;
END_IF
END_FUNCTION

(* ---------- FC_HeatColor:热力色阶(C2/C6,0711) ----------
   值→蓝(冷)→黄(中)→红(热)三段线性插值,工业监控惯例。
   端点:0=16#FF1565C0 蓝 / 0.5=16#FFFFD600 黄 / 1=16#FFE53935 红;rMax<=0 返回蓝(防除)。
   RGBA 前导 FF=不透明(0710 实证:00 前缀渲染全透明)。 *)
FUNCTION FC_HeatColor : DWORD
VAR_INPUT
    rVal : REAL;
    rMax : REAL;
END_VAR
VAR
    rT, rSeg : REAL;       // 勿用 t/d 等单字母(TIME/DATE 字面量前缀保留,同 0706 r/s 教训)
    iR, iG, iB : INT;
END_VAR
IF rMax <= 0.0 THEN
    FC_HeatColor := 16#FF1565C0;  RETURN;
END_IF
rT := rVal / rMax;
IF rT < 0.0 THEN rT := 0.0; END_IF
IF rT > 1.0 THEN rT := 1.0; END_IF
IF rT < 0.5 THEN
    rSeg := rT * 2.0;                            // 蓝(21,101,192)→黄(255,214,0)
    iR := REAL_TO_INT(21.0  + (255.0 - 21.0)  * rSeg);
    iG := REAL_TO_INT(101.0 + (214.0 - 101.0) * rSeg);
    iB := REAL_TO_INT(192.0 + (0.0   - 192.0) * rSeg);
ELSE
    rSeg := (rT - 0.5) * 2.0;                    // 黄(255,214,0)→红(229,57,53)
    iR := REAL_TO_INT(255.0 + (229.0 - 255.0) * rSeg);
    iG := REAL_TO_INT(214.0 + (57.0  - 214.0) * rSeg);
    iB := REAL_TO_INT(0.0   + (53.0  - 0.0)   * rSeg);
END_IF
FC_HeatColor := 16#FF000000
    OR SHL(INT_TO_DWORD(iR), 16) OR SHL(INT_TO_DWORD(iG), 8) OR INT_TO_DWORD(iB);
END_FUNCTION

(* ---------- FC_BlendLight:向白混色 45%(C1 层高亮,0711) ----------
   任意底色(状态/热力)上的选中层加亮通道:每通道 c := c + (255-c)*0.45。 *)
FUNCTION FC_BlendLight : DWORD
VAR_INPUT
    dw : DWORD;
END_VAR
VAR
    iR, iG, iB : INT;
END_VAR
iR := DWORD_TO_INT(SHR(dw, 16) AND 16#FF);
iG := DWORD_TO_INT(SHR(dw, 8) AND 16#FF);
iB := DWORD_TO_INT(dw AND 16#FF);
iR := REAL_TO_INT(INT_TO_REAL(iR) + (255.0 - INT_TO_REAL(iR)) * 0.45);
iG := REAL_TO_INT(INT_TO_REAL(iG) + (255.0 - INT_TO_REAL(iG)) * 0.45);
iB := REAL_TO_INT(INT_TO_REAL(iB) + (255.0 - INT_TO_REAL(iB)) * 0.45);
FC_BlendLight := 16#FF000000
    OR SHL(INT_TO_DWORD(iR), 16) OR SHL(INT_TO_DWORD(iG), 8) OR INT_TO_DWORD(iB);
END_FUNCTION

(* ---------- FC_TravelLaden:载货行程时间(U2 载重运动学,块3 拟真对照) ----------
   功能:垂直轴速度 × GVL_Param.rLadenFactorVY(满载折减,默认0.80),水平不折减;
        xUseAccel/xSimXY 开关行为与 FC_CalcTravelTime 完全同构(sim travel_time_laden 一字对齐)。
   输入:x0,y0,x1,y1 格坐标;xSimXY TRUE=切比雪夫 FALSE=顺序模型
   输出:载货行程时间 s(纯行程,不含装卸——装卸另用 FC_HandleTime,避免双计 rTLoad)
   边界:速度/折减系数非法(<=0)钳回安全值;dx/dy 由 ABS 保证非负
   示例:laden(0,0→10,10) 主口径 vy=0.5×0.8=0.4 → MAX(10/2, 10/0.4)=25.0s(空载 20.0s,T45 锚)
   消费:FB_QueryGood(QryTravelLaden);不进评分/分配链路(零回归设计) *)
FUNCTION FC_TravelLaden : REAL
VAR_INPUT
    x0, y0, x1, y1  : INT;      // 起点/终点(格坐标)
    xSimXY          : BOOL;     // TRUE=切比雪夫 FALSE=顺序
END_VAR
VAR
    dx, dy, tx, ty : REAL;
    vx, vy         : REAL;
END_VAR
dx := ABS(INT_TO_REAL(x1 - x0)) * GVL_Param.CELL_W;
dy := ABS(INT_TO_REAL(y1 - y0)) * GVL_Param.CELL_H;
// 边界:速度与折减系数非法保护(调参区可被改出非法值,拒绝依赖画面侧校验)
vx := GVL_Param.rVx;  IF vx <= 0.0 THEN vx := 1.0; END_IF
vy := GVL_Param.rVy;  IF vy <= 0.0 THEN vy := 1.0; END_IF
IF GVL_Param.rLadenFactorVY > 0.0 AND GVL_Param.rLadenFactorVY <= 1.0 THEN
    vy := vy * GVL_Param.rLadenFactorVY;    // 满载垂直折减(仅垂直,U2 口径)
END_IF
IF GVL_Param.xUseAccel THEN
    tx := FC_AxisTime(d := dx, vmax := vx, acc := GVL_Param.rAx);
    ty := FC_AxisTime(d := dy, vmax := vy, acc := GVL_Param.rAy);
ELSE
    tx := dx / vx;
    ty := dy / vy;
END_IF
IF xSimXY THEN
    FC_TravelLaden := MAX(tx, ty);
ELSE
    FC_TravelLaden := tx + ty;
END_IF
END_FUNCTION

(* ---------- FC_HandleTime:装卸时间三档(U2 可变装卸,块3 拟真对照) ----------
   功能:按货物重量查三档装卸时长(轻<=W1→T1 / 中<=W2→T2 / 重>W2→T3);
        档界与时长全部 GVL_Param 参数化 = 画面调参区旋钮(改档界/时长,查询页数字实时变)。
   输入:rW 货物重量 kg(定义域>=0;负值落轻货档,入口校验由 FB_GoodsInput iErrId=2 兜底)
   输出:单次装卸时间 s(货叉全循环;sim handle_time 一字对齐,默认档 6.0/8.5/12.5)
   边界:档界被调成 W1>W2 时按 ELSIF 顺序自然判定(W1 优先),无崩溃路径
   示例:29.9→6.0 / 30.1→8.5 / 60.1→12.5(T44 三档边界锚,0.1 间隙避单精度) *)
FUNCTION FC_HandleTime : REAL
VAR_INPUT
    rW : REAL;                  // 货物重量 kg
END_VAR
IF rW <= GVL_Param.rHandleW1 THEN
    FC_HandleTime := GVL_Param.rHandleT1;
ELSIF rW <= GVL_Param.rHandleW2 THEN
    FC_HandleTime := GVL_Param.rHandleT2;
ELSE
    FC_HandleTime := GVL_Param.rHandleT3;
END_IF
END_FUNCTION

(* ---- 04_FB_Warehouse.st ---- *)
(* ============================================================
   04_FB_Warehouse.st — 功能块(FB,有状态)
   导入方法:每个 FUNCTION_BLOCK 建一个 POU(类型"功能块"),粘贴对应段落
   核心设计:扫描周期感知的分片执行 —— 批量分配与局部搜索都做成
   跨周期状态机,每个扫描周期只处理有限计算量(GVL_Param.nBatchPerCycle/
   nPairsPerCycle),不阻塞、不触发看门狗;xBusy/xDone 汇报进度。
   这是本方案的 PLC 原生工程点:优化算法以非阻塞方式跑在实时控制器上。
   ============================================================ *)

(* ---------- FB_InitWarehouse:初始化仓库(单周期) ---------- *)
FUNCTION_BLOCK FB_InitWarehouse
VAR_INPUT
    xExecute : BOOL;            // 上升沿触发
    iRule    : INT;             // 预占用解读(B1)
END_VAR
VAR_OUTPUT
    xDone     : BOOL;
    iPreCount : INT;            // 预占用格数(rule3=133官方/rule0=49/rule1=231/rule2=134,自检用)
END_VAR
VAR
    xOld : BOOL;
    x, y : INT;
END_VAR

IF xExecute AND NOT xOld THEN
    iPreCount := 0;
    FOR x := 0 TO GVL_Param.COLS - 1 DO
        FOR y := 0 TO GVL_Param.TIERS - 1 DO
            GVL_WH.aSlots[x, y].X         := x;
            GVL_WH.aSlots[x, y].Y         := y;
            GVL_WH.aSlots[x, y].CapCoef   := FC_CapCoef(y := y);
            GVL_WH.aSlots[x, y].MaxWeight := GVL_WH.aSlots[x, y].CapCoef * GVL_Param.BASE_CAP;
            GVL_WH.aSlots[x, y].MaxVolume := GVL_Param.CELL_VOL;
            GVL_WH.aSlots[x, y].PresetOcc := FC_IsPresetOccupied(x := x, y := y, iRule := iRule);
            GVL_WH.aSlots[x, y].Occupied  := GVL_WH.aSlots[x, y].PresetOcc;
            GVL_WH.aSlots[x, y].GoodsId   := 0;
            GVL_WH.aSlotFreq[x, y]        := 0.0;    // C2 布局态随批清;aSlotOps 履历不清(C6)
            IF GVL_WH.aSlots[x, y].PresetOcc THEN
                iPreCount := iPreCount + 1;
                GVL_Visu.VisuSlotState[x, y] := 1;   // 深灰:预占用
            ELSE
                GVL_Visu.VisuSlotState[x, y] := 0;   // 浅灰:空闲
            END_IF
        END_FOR
    END_FOR
    xDone := TRUE;
END_IF
// 0711 修:完成即撤沿。本 FB 是"单拍完成+完成拍输入仍 TRUE+完成后停止调用"模式,
// 旧写法 xOld:=xExecute 会把 xOld 冻结在 TRUE,Reset 二次进入时沿失效→仓库不重建、
// xDone 残留 TRUE 令状态机瞬转(实测:Reset 后 aSlots 旧占位残留/统计跳算的根因之一)。
xOld := xExecute AND NOT xDone;
END_FUNCTION_BLOCK

(* ---------- FB_SelectSlot:单件货选位(单周期,400 仓位全扫描) ----------
   iStrategy: 0=seq 首个可行位(题面"连续存放"字面基线)
              1=near 行程时间最小
              2=score 多目标评分最小(主线)
   扫描顺序 x外层/y内层,平局保留先者 —— 与 Python 迭代序/tie-break 一字对齐 *)
FUNCTION_BLOCK FB_SelectSlot
VAR_INPUT
    iStrategy : INT;
    rGoodW    : REAL;
    rGoodF    : REAL;
    rGoodV    : REAL;
    rWMax     : REAL;           // 批次归一分母(由调用方维护)
    rFMax     : REAL;
END_VAR
VAR_OUTPUT
    xFound     : BOOL;
    iBestX     : INT;
    iBestY     : INT;
    rBestScore : REAL;
    rBestTime  : REAL;
END_VAR
VAR
    x, y      : INT;
    rS, rT    : REAL;
    xBetter   : BOOL;
END_VAR

xFound := FALSE;
iBestX := -1;  iBestY := -1;
rBestScore := 3.4E38;  rBestTime := 3.4E38;

FOR x := 0 TO GVL_Param.COLS - 1 DO
    FOR y := 0 TO GVL_Param.TIERS - 1 DO
        IF FC_CheckFeasible(x := x, y := y, rGoodW := rGoodW, rGoodV := rGoodV) THEN
            IF iStrategy = 0 THEN
                // seq:第一个可行位即返回
                xFound := TRUE;  iBestX := x;  iBestY := y;
                rBestTime  := FC_CalcTravelTime(x0 := 0, y0 := 0, x1 := x, y1 := y,
                                                xSimXY := GVL_Param.xSimultaneousXY);
                rBestScore := FC_CalcScore(rGoodW := rGoodW, rGoodF := rGoodF, x := x, y := y,
                                           rWMax := rWMax, rFMax := rFMax);
                RETURN;
            END_IF
            rT := FC_CalcTravelTime(x0 := 0, y0 := 0, x1 := x, y1 := y,
                                    xSimXY := GVL_Param.xSimultaneousXY);
            IF iStrategy = 1 THEN
                // near:按 (时间, 层, 列) 严格更小才替换(平局保先者=Python min 语义)
                xBetter := rT < rBestTime;
            ELSE
                // score:按 (评分, 时间) 严格更小;层/列由扫描顺序天然兜底
                rS := FC_CalcScore(rGoodW := rGoodW, rGoodF := rGoodF, x := x, y := y,
                                   rWMax := rWMax, rFMax := rFMax);
                xBetter := (rS < rBestScore) OR ((rS = rBestScore) AND (rT < rBestTime));
            END_IF
            IF xBetter THEN
                xFound := TRUE;  iBestX := x;  iBestY := y;  rBestTime := rT;
                IF iStrategy = 2 THEN rBestScore := rS;
                ELSE rBestScore := FC_CalcScore(rGoodW := rGoodW, rGoodF := rGoodF,
                                                x := x, y := y, rWMax := rWMax, rFMax := rFMax);
                END_IF
            END_IF
        END_IF
    END_FOR
END_FOR
END_FUNCTION_BLOCK

(* ---------- FB_AssignAllGoods:批量分配(分片状态机,跨扫描周期) ----------
   xUseRank=TRUE  → AWRA 模式:先按优先级排序(重货/高频先挑),再逐件选位
   xUseRank=FALSE → 在线模式:按到达顺序逐件选位(决赛交互场景等价)
   每周期只处理 nBatchPerCycle 件(排序阶段每周期 nSortOuter 个外层位),非阻塞 *)
FUNCTION_BLOCK FB_AssignAllGoods
VAR_INPUT
    xStart    : BOOL;           // 上升沿启动
    xUseRank  : BOOL;
    iStrategy : INT;            // 传给 FB_SelectSlot(0/1/2)
END_VAR
VAR_OUTPUT
    xBusy     : BOOL;
    xDone     : BOOL;
    iAssigned : INT;
    iFailed   : INT;
END_VAR
VAR
    xOld       : BOOL;
    iPhase     : INT;           // 0=空闲 1=算优先级+初始化索引 2=排序 3=分配 4=完成
    i, j, k    : INT;
    iCur       : INT;           // 分配游标(在 aRankIdx 上)
    iSortPos   : INT;           // 选择排序外层游标
    nSortOuter : INT := 20;     // 排序阶段每周期处理的外层位数
    iBestJ     : INT;
    iTmp       : INT;
    rWMax, rFMax, rVMax : REAL;
    fbSel      : FB_SelectSlot;
    iG         : INT;
END_VAR

IF xStart AND NOT xOld THEN
    IF GVL_WH.iGoodsCount > 0 THEN
        iPhase := 1;  xBusy := TRUE;  xDone := FALSE;
        iAssigned := 0;  iFailed := 0;  iCur := 1;  iSortPos := 1;
    END_IF
END_IF
xOld := xStart;

CASE iPhase OF
    1:  // ---- 归一分母 + 优先级 + 索引初始化(单周期,O(n)) ----
        rWMax := 0.0;  rFMax := 0.0;  rVMax := 0.0;
        FOR i := 1 TO GVL_WH.iGoodsCount DO
            IF GVL_WH.aGoods[i].Weight > rWMax THEN rWMax := GVL_WH.aGoods[i].Weight; END_IF
            IF GVL_WH.aGoods[i].Freq   > rFMax THEN rFMax := GVL_WH.aGoods[i].Freq;   END_IF
            IF GVL_WH.aGoods[i].Volume > rVMax THEN rVMax := GVL_WH.aGoods[i].Volume; END_IF
        END_FOR
        FOR i := 1 TO GVL_WH.iGoodsCount DO
            GVL_WH.aRankIdx[i] := i;
            GVL_WH.aGoods[i].Priority := FC_CalcPriority(
                rGoodF := GVL_WH.aGoods[i].Freq,  rGoodW := GVL_WH.aGoods[i].Weight,
                rGoodV := GVL_WH.aGoods[i].Volume,
                rFMax := rFMax, rWMax := rWMax, rVMax := rVMax);
        END_FOR
        IF xUseRank THEN iPhase := 2; ELSE iPhase := 3; END_IF

    2:  // ---- Rank:选择排序(优先级降序,平局按Id升序;分片:每周期 nSortOuter 位) ----
        k := 0;
        WHILE (k < nSortOuter) AND (iSortPos < GVL_WH.iGoodsCount) DO
            iBestJ := iSortPos;
            FOR j := iSortPos + 1 TO GVL_WH.iGoodsCount DO
                IF (GVL_WH.aGoods[GVL_WH.aRankIdx[j]].Priority >
                    GVL_WH.aGoods[GVL_WH.aRankIdx[iBestJ]].Priority)
                OR ((GVL_WH.aGoods[GVL_WH.aRankIdx[j]].Priority =
                     GVL_WH.aGoods[GVL_WH.aRankIdx[iBestJ]].Priority)
                    AND (GVL_WH.aRankIdx[j] < GVL_WH.aRankIdx[iBestJ])) THEN
                    iBestJ := j;
                END_IF
            END_FOR
            iTmp := GVL_WH.aRankIdx[iSortPos];
            GVL_WH.aRankIdx[iSortPos] := GVL_WH.aRankIdx[iBestJ];
            GVL_WH.aRankIdx[iBestJ]   := iTmp;
            iSortPos := iSortPos + 1;
            k := k + 1;
        END_WHILE
        IF iSortPos >= GVL_WH.iGoodsCount THEN iPhase := 3; END_IF

    3:  // ---- Assign:逐件选位(分片:每周期 nBatchPerCycle 件) ----
        k := 0;
        WHILE (k < GVL_Param.nBatchPerCycle) AND (iCur <= GVL_WH.iGoodsCount) DO
            iG := GVL_WH.aRankIdx[iCur];
            fbSel(iStrategy := iStrategy,
                  rGoodW := GVL_WH.aGoods[iG].Weight,
                  rGoodF := GVL_WH.aGoods[iG].Freq,
                  rGoodV := GVL_WH.aGoods[iG].Volume,
                  rWMax := rWMax, rFMax := rFMax);
            IF fbSel.xFound THEN
                GVL_WH.aSlots[fbSel.iBestX, fbSel.iBestY].Occupied := TRUE;
                GVL_WH.aSlots[fbSel.iBestX, fbSel.iBestY].GoodsId  := GVL_WH.aGoods[iG].Id;
                GVL_WH.aSlotFreq[fbSel.iBestX, fbSel.iBestY] := GVL_WH.aGoods[iG].Freq;   // C2
                GVL_WH.aSlotOps[fbSel.iBestX, fbSel.iBestY] := GVL_WH.aSlotOps[fbSel.iBestX, fbSel.iBestY] + 1;  // C6 履历
                GVL_WH.aGoods[iG].Assigned   := TRUE;
                GVL_WH.aGoods[iG].X          := fbSel.iBestX;
                GVL_WH.aGoods[iG].Y          := fbSel.iBestY;
                GVL_WH.aGoods[iG].Score      := fbSel.rBestScore;
                GVL_WH.aGoods[iG].ExecTime   := fbSel.rBestTime;
                GVL_WH.aGoods[iG].PathLength := FC_CalcPathLen(x0 := 0, y0 := 0,
                                                x1 := fbSel.iBestX, y1 := fbSel.iBestY);
                GVL_Visu.VisuSlotState[fbSel.iBestX, fbSel.iBestY] := 2;   // 绿:已占
                iAssigned := iAssigned + 1;
            ELSE
                // 边界:无可行位 → 计数并报警文本(边界清单#9)
                GVL_WH.aGoods[iG].Assigned := FALSE;
                GVL_WH.aGoods[iG].X := -1;  GVL_WH.aGoods[iG].Y := -1;
                iFailed := iFailed + 1;
                GVL_Visu.VisuStatusText := CONCAT('NO_SLOT_GOODS_ID=',
                                                  INT_TO_STRING(GVL_WH.aGoods[iG].Id));
            END_IF
            iCur := iCur + 1;
            k := k + 1;
        END_WHILE
        IF iCur > GVL_WH.iGoodsCount THEN iPhase := 4; END_IF

    4:  // ---- 完成 ----
        xBusy := FALSE;  xDone := TRUE;  iPhase := 0;
END_CASE
END_FUNCTION_BLOCK

(* ---------- FB_LocalSwapImprove:局部搜索(AWRA-LS 第三段,分片状态机) ----------
   每轮 = 重定位阶段(逐货找更优空位)+ 成对交换阶段(互换后总分下降则换);
   有改进继续下一轮(≤nMaxLsRounds),无改进提前收敛。
   一切换位前重查物理约束(FC_FitsPhysical,边界清单#10)。 *)
FUNCTION_BLOCK FB_LocalSwapImprove
VAR_INPUT
    xStart : BOOL;
END_VAR
VAR_OUTPUT
    xBusy   : BOOL;
    xDone   : BOOL;
    iSwaps  : INT;
    iRelocs : INT;
    iRounds : INT;
END_VAR
VAR
    xOld       : BOOL;
    iPhase     : INT;           // 0=空闲 1=重定位 2=交换 3=轮末判定 4=完成
    xImproved  : BOOL;
    iCurR      : INT;           // 重定位游标(aRankIdx 序,与 Python 一致)
    iI, iJ     : INT;           // 交换双游标(i<j)
    k, x, y    : INT;
    iGi, iGj   : INT;
    rWMax, rFMax : REAL;
    i          : INT;
    rCur, rBest, rS, rOld, rNew : REAL;
    iBx, iBy   : INT;
    xiA, yiA, xjA, yjA : INT;
END_VAR

IF xStart AND NOT xOld THEN
    IF GVL_WH.iGoodsCount > 0 THEN
        // 归一分母与分配阶段口径一致
        rWMax := 0.0;  rFMax := 0.0;
        FOR i := 1 TO GVL_WH.iGoodsCount DO
            IF GVL_WH.aGoods[i].Weight > rWMax THEN rWMax := GVL_WH.aGoods[i].Weight; END_IF
            IF GVL_WH.aGoods[i].Freq   > rFMax THEN rFMax := GVL_WH.aGoods[i].Freq;   END_IF
        END_FOR
        iPhase := 1;  xBusy := TRUE;  xDone := FALSE;
        iSwaps := 0;  iRelocs := 0;  iRounds := 1;  xImproved := FALSE;
        iCurR := 1;  iI := 1;  iJ := 2;
    END_IF
END_IF
xOld := xStart;

CASE iPhase OF
    1:  // ---- 重定位:每周期 nBatchPerCycle 件,每件全库扫描更优空位 ----
        k := 0;
        WHILE (k < GVL_Param.nBatchPerCycle) AND (iCurR <= GVL_WH.iGoodsCount) DO
            iGi := GVL_WH.aRankIdx[iCurR];
            IF GVL_WH.aGoods[iGi].Assigned THEN
                rCur := FC_CalcScore(rGoodW := GVL_WH.aGoods[iGi].Weight,
                                     rGoodF := GVL_WH.aGoods[iGi].Freq,
                                     x := GVL_WH.aGoods[iGi].X, y := GVL_WH.aGoods[iGi].Y,
                                     rWMax := rWMax, rFMax := rFMax);
                rBest := rCur;  iBx := -1;  iBy := -1;
                FOR x := 0 TO GVL_Param.COLS - 1 DO
                    FOR y := 0 TO GVL_Param.TIERS - 1 DO
                        IF FC_CheckFeasible(x := x, y := y,
                                            rGoodW := GVL_WH.aGoods[iGi].Weight,
                                            rGoodV := GVL_WH.aGoods[iGi].Volume) THEN
                            rS := FC_CalcScore(rGoodW := GVL_WH.aGoods[iGi].Weight,
                                               rGoodF := GVL_WH.aGoods[iGi].Freq,
                                               x := x, y := y, rWMax := rWMax, rFMax := rFMax);
                            IF rS < rBest - 0.000001 THEN
                                rBest := rS;  iBx := x;  iBy := y;
                            END_IF
                        END_IF
                    END_FOR
                END_FOR
                IF iBx >= 0 THEN
                    // 搬移:旧位腾空,新位占用,货物记录/可视化联动
                    GVL_WH.aSlots[GVL_WH.aGoods[iGi].X, GVL_WH.aGoods[iGi].Y].Occupied := FALSE;
                    GVL_WH.aSlots[GVL_WH.aGoods[iGi].X, GVL_WH.aGoods[iGi].Y].GoodsId  := 0;
                    GVL_WH.aSlotFreq[GVL_WH.aGoods[iGi].X, GVL_WH.aGoods[iGi].Y] := 0.0;   // C2 腾空
                    GVL_Visu.VisuSlotState[GVL_WH.aGoods[iGi].X, GVL_WH.aGoods[iGi].Y] := 0;
                    GVL_WH.aSlots[iBx, iBy].Occupied := TRUE;
                    GVL_WH.aSlots[iBx, iBy].GoodsId  := GVL_WH.aGoods[iGi].Id;
                    GVL_WH.aSlotFreq[iBx, iBy] := GVL_WH.aGoods[iGi].Freq;                 // C2
                    GVL_WH.aSlotOps[iBx, iBy] := GVL_WH.aSlotOps[iBx, iBy] + 1;            // C6 搬移=一次存取
                    GVL_Visu.VisuSlotState[iBx, iBy] := 2;
                    GVL_WH.aGoods[iGi].X := iBx;  GVL_WH.aGoods[iGi].Y := iBy;
                    GVL_WH.aGoods[iGi].Score := rBest;
                    GVL_WH.aGoods[iGi].ExecTime := FC_CalcTravelTime(x0 := 0, y0 := 0,
                                        x1 := iBx, y1 := iBy, xSimXY := GVL_Param.xSimultaneousXY);
                    GVL_WH.aGoods[iGi].PathLength := FC_CalcPathLen(x0 := 0, y0 := 0, x1 := iBx, y1 := iBy);
                    iRelocs := iRelocs + 1;  xImproved := TRUE;
                END_IF
            END_IF
            iCurR := iCurR + 1;  k := k + 1;
        END_WHILE
        IF iCurR > GVL_WH.iGoodsCount THEN
            iPhase := 2;  iI := 1;  iJ := 2;
        END_IF

    2:  // ---- 成对交换:每周期 nPairsPerCycle 对 ----
        k := 0;
        WHILE (k < GVL_Param.nPairsPerCycle) AND (iI < GVL_WH.iGoodsCount) DO
            iGi := GVL_WH.aRankIdx[iI];  iGj := GVL_WH.aRankIdx[iJ];
            IF GVL_WH.aGoods[iGi].Assigned AND GVL_WH.aGoods[iGj].Assigned THEN
                xiA := GVL_WH.aGoods[iGi].X;  yiA := GVL_WH.aGoods[iGi].Y;
                xjA := GVL_WH.aGoods[iGj].X;  yjA := GVL_WH.aGoods[iGj].Y;
                // 换位前双向物理约束复查(承重/容积)
                IF FC_FitsPhysical(x := xjA, y := yjA, rGoodW := GVL_WH.aGoods[iGi].Weight,
                                   rGoodV := GVL_WH.aGoods[iGi].Volume)
                AND FC_FitsPhysical(x := xiA, y := yiA, rGoodW := GVL_WH.aGoods[iGj].Weight,
                                    rGoodV := GVL_WH.aGoods[iGj].Volume) THEN
                    rOld := FC_CalcScore(rGoodW := GVL_WH.aGoods[iGi].Weight, rGoodF := GVL_WH.aGoods[iGi].Freq,
                                         x := xiA, y := yiA, rWMax := rWMax, rFMax := rFMax)
                          + FC_CalcScore(rGoodW := GVL_WH.aGoods[iGj].Weight, rGoodF := GVL_WH.aGoods[iGj].Freq,
                                         x := xjA, y := yjA, rWMax := rWMax, rFMax := rFMax);
                    rNew := FC_CalcScore(rGoodW := GVL_WH.aGoods[iGi].Weight, rGoodF := GVL_WH.aGoods[iGi].Freq,
                                         x := xjA, y := yjA, rWMax := rWMax, rFMax := rFMax)
                          + FC_CalcScore(rGoodW := GVL_WH.aGoods[iGj].Weight, rGoodF := GVL_WH.aGoods[iGj].Freq,
                                         x := xiA, y := yiA, rWMax := rWMax, rFMax := rFMax);
                    IF rNew < rOld - 0.000001 THEN
                        GVL_WH.aSlots[xiA, yiA].GoodsId := GVL_WH.aGoods[iGj].Id;
                        GVL_WH.aSlots[xjA, yjA].GoodsId := GVL_WH.aGoods[iGi].Id;
                        GVL_WH.aSlotFreq[xiA, yiA] := GVL_WH.aGoods[iGj].Freq;   // C2 互换
                        GVL_WH.aSlotFreq[xjA, yjA] := GVL_WH.aGoods[iGi].Freq;
                        GVL_WH.aSlotOps[xiA, yiA] := GVL_WH.aSlotOps[xiA, yiA] + 1;  // C6 交换=两格各一次存取
                        GVL_WH.aSlotOps[xjA, yjA] := GVL_WH.aSlotOps[xjA, yjA] + 1;
                        GVL_WH.aGoods[iGi].X := xjA;  GVL_WH.aGoods[iGi].Y := yjA;
                        GVL_WH.aGoods[iGj].X := xiA;  GVL_WH.aGoods[iGj].Y := yiA;
                        GVL_WH.aGoods[iGi].ExecTime := FC_CalcTravelTime(x0 := 0, y0 := 0,
                                            x1 := xjA, y1 := yjA, xSimXY := GVL_Param.xSimultaneousXY);
                        GVL_WH.aGoods[iGj].ExecTime := FC_CalcTravelTime(x0 := 0, y0 := 0,
                                            x1 := xiA, y1 := yiA, xSimXY := GVL_Param.xSimultaneousXY);
                        GVL_WH.aGoods[iGi].PathLength := FC_CalcPathLen(x0 := 0, y0 := 0, x1 := xjA, y1 := yjA);
                        GVL_WH.aGoods[iGj].PathLength := FC_CalcPathLen(x0 := 0, y0 := 0, x1 := xiA, y1 := yiA);
                        iSwaps := iSwaps + 1;  xImproved := TRUE;
                    END_IF
                END_IF
            END_IF
            // 游标推进(i<j 上三角遍历)
            iJ := iJ + 1;
            IF iJ > GVL_WH.iGoodsCount THEN
                iI := iI + 1;  iJ := iI + 1;
            END_IF
            k := k + 1;
        END_WHILE
        IF iI >= GVL_WH.iGoodsCount THEN iPhase := 3; END_IF

    3:  // ---- 轮末判定 ----
        IF xImproved AND (iRounds < GVL_Param.nMaxLsRounds) THEN
            iRounds := iRounds + 1;  xImproved := FALSE;
            iCurR := 1;  iPhase := 1;               // 下一轮从重定位开始
        ELSE
            iPhase := 4;
        END_IF

    4:  // ---- 完成 ----
        xBusy := FALSE;  xDone := TRUE;  iPhase := 0;
END_CASE
END_FUNCTION_BLOCK

(* ---------- FB_Stats:统计计算(单周期;口径C1-C8,与 Python metrics 对齐) ---------- *)
FUNCTION_BLOCK FB_Stats
VAR_INPUT
    xExecute : BOOL;
END_VAR
VAR_OUTPUT
    xDone : BOOL;
END_VAR
VAR
    xOld : BOOL;
    i, x, y, nUsed : INT;
    rT, rFSum, rWSum, rFT, rWH : REAL;
END_VAR

IF xExecute AND NOT xOld THEN
    GVL_WH.stStats.PlacedCnt := 0;   GVL_WH.stStats.FailedCnt := 0;
    GVL_WH.stStats.TotalTime2Way := 0.0;  GVL_WH.stStats.PathTotal2Way := 0.0;
    GVL_WH.stStats.Energy := 0.0;    GVL_WH.stStats.ViolCnt := 0;
    rFSum := 0.0;  rWSum := 0.0;  rFT := 0.0;  rWH := 0.0;

    FOR i := 1 TO GVL_WH.iGoodsCount DO
        IF GVL_WH.aGoods[i].Assigned THEN
            GVL_WH.stStats.PlacedCnt := GVL_WH.stStats.PlacedCnt + 1;
            rT := GVL_WH.aGoods[i].ExecTime;
            GVL_WH.stStats.TotalTime2Way  := GVL_WH.stStats.TotalTime2Way  + 2.0 * rT;
            GVL_WH.stStats.PathTotal2Way  := GVL_WH.stStats.PathTotal2Way  + 2.0 * GVL_WH.aGoods[i].PathLength;
            rFSum := rFSum + GVL_WH.aGoods[i].Freq;
            rFT   := rFT   + GVL_WH.aGoods[i].Freq * rT;
            rWSum := rWSum + GVL_WH.aGoods[i].Weight;
            rWH   := rWH   + GVL_WH.aGoods[i].Weight * INT_TO_REAL(GVL_WH.aGoods[i].Y) * GVL_Param.CELL_H;
            // C8 违规复查:分配结果必须仍满足约束(恒0,非0=程序缺陷立即可见)
            IF (GVL_WH.aGoods[i].Weight > GVL_WH.aSlots[GVL_WH.aGoods[i].X, GVL_WH.aGoods[i].Y].MaxWeight)
            OR (GVL_WH.aGoods[i].Volume > GVL_WH.aSlots[GVL_WH.aGoods[i].X, GVL_WH.aGoods[i].Y].MaxVolume) THEN
                GVL_WH.stStats.ViolCnt := GVL_WH.stStats.ViolCnt + 1;
            END_IF
        ELSE
            GVL_WH.stStats.FailedCnt := GVL_WH.stStats.FailedCnt + 1;
        END_IF
    END_FOR

    IF GVL_WH.stStats.PlacedCnt > 0 THEN
        GVL_WH.stStats.AvgTime := GVL_WH.stStats.TotalTime2Way / INT_TO_REAL(GVL_WH.stStats.PlacedCnt);
    ELSE
        GVL_WH.stStats.AvgTime := 0.0;
    END_IF
    IF rFSum > 0.0 THEN GVL_WH.stStats.ExpRetrieval := rFT / rFSum; ELSE GVL_WH.stStats.ExpRetrieval := 0.0; END_IF
    IF rWSum > 0.0 THEN GVL_WH.stStats.CogHeight := rWH / rWSum;    ELSE GVL_WH.stStats.CogHeight := 0.0;    END_IF
    GVL_WH.stStats.Energy := rWH;                       // Σ 重量*高度 kg·m(C4)

    nUsed := 0;
    FOR x := 0 TO GVL_Param.COLS - 1 DO
        FOR y := 0 TO GVL_Param.TIERS - 1 DO
            IF GVL_WH.aSlots[x, y].Occupied THEN nUsed := nUsed + 1; END_IF
        END_FOR
    END_FOR
    GVL_WH.stStats.UtilPct := INT_TO_REAL(nUsed) / INT_TO_REAL(GVL_Param.COLS * GVL_Param.TIERS);

    // 同步可视化统计区
    GVL_Visu.VisuTotalTime := GVL_WH.stStats.TotalTime2Way;
    GVL_Visu.VisuAvgTime   := GVL_WH.stStats.AvgTime;
    GVL_Visu.VisuSpaceUtilization := GVL_WH.stStats.UtilPct;
    GVL_Visu.VisuViolationCount   := GVL_WH.stStats.ViolCnt;
    xDone := TRUE;
END_IF
// 0711 修:完成即撤沿(同 FB_InitWarehouse)。旧写法在"单拍完成+完成拍 xExecute=TRUE+
// 完成后不再被调用"下冻结 xOld→第二次批量统计跳算,显示残留 Reset 清的 0(实测复现)。
xOld := xExecute AND NOT xDone;
END_FUNCTION_BLOCK

(* ---------- FB_AnimatePath:堆垛机动画回放(L6 决赛可视化核心) ----------
   沿 VisuPath 的 L 形物理走线逐点推进 VisuCurrentX/Y,总时长 = 该点切比雪夫
   行程时间 × 回放倍率(口径 C2:显示走线为曼哈顿,时序按切比雪夫等比回放,
   两口径并列的动画化呈现)。先调 FB_BuildVisuPath 生成路径再启动本 FB。 *)
FUNCTION_BLOCK FB_AnimatePath
VAR_INPUT
    xStart      : BOOL;         // 上升沿启动回放
    rCycleTime  : REAL := 0.01; // 本任务周期 s(10ms 任务填 0.01)
    rSpeedScale : REAL := 5.0;  // 回放倍速(5=五倍速演示)
END_VAR
VAR_OUTPUT
    xBusy : BOOL;
    xDone : BOOL;
END_VAR
VAR
    xOld     : BOOL;
    rElapsed : REAL;            // 已回放的"仿真时间" s
    rTotal   : REAL;            // 目标点切比雪夫总时长 s
    iIdx     : INT;
END_VAR

IF xStart AND NOT xOld THEN
    IF GVL_Visu.VisuPathCount > 1 THEN
        rTotal := FC_CalcTravelTime(x0 := 0, y0 := 0,
                                    x1 := GVL_Visu.VisuTargetX, y1 := GVL_Visu.VisuTargetY,
                                    xSimXY := GVL_Param.xSimultaneousXY);
        IF rTotal <= 0.0 THEN rTotal := 0.001; END_IF
        rElapsed := 0.0;  xBusy := TRUE;  xDone := FALSE;
        GVL_Visu.VisuCurrentX := GVL_Visu.VisuPathX[0];
        GVL_Visu.VisuCurrentY := GVL_Visu.VisuPathY[0];
    END_IF
END_IF
xOld := xStart;

IF xBusy THEN
    IF GVL_Visu.VisuPathCount < 2 THEN
        // 回放途中路径被外部清除(复位/批量启动会清 VisuPathCount)→ 中止,
        // 否则下面 PathCount-1 = -1 会造成数组负索引越界(真实边界,勿删护栏)
        xBusy := FALSE;  xDone := TRUE;
    ELSE
        rElapsed := rElapsed + rCycleTime * rSpeedScale;
        // 路径索引 = 已过时间占比 × 路径点数(线性等比映射)
        iIdx := REAL_TO_INT(rElapsed / rTotal * INT_TO_REAL(GVL_Visu.VisuPathCount - 1));
        IF iIdx >= GVL_Visu.VisuPathCount - 1 THEN
            iIdx := GVL_Visu.VisuPathCount - 1;
            xBusy := FALSE;  xDone := TRUE;
        END_IF
        GVL_Visu.VisuCurrentX := GVL_Visu.VisuPathX[iIdx];
        GVL_Visu.VisuCurrentY := GVL_Visu.VisuPathY[iIdx];
    END_IF
END_IF
END_FUNCTION_BLOCK

(* ---------- FB_ScanLoadProbe:L4 扫描周期负载实测(AC500 实现章的实测数据源) ----------
   用法:在要测量的代码段前后各调一次:
     fbProbe(xStart := TRUE);   (* 段前 *)
     ... 被测代码(如 fbAssign 一个分片周期)...
     fbProbe(xStop := TRUE);    (* 段后 *)
   输出微秒级 单次/平均/最大 耗时与样本数 —— 报告里给出
   "10ms 任务周期下分片计算占用 X%(看门狗裕量 Y 倍)"的实测表。 *)
FUNCTION_BLOCK FB_ScanLoadProbe
VAR_INPUT
    xStart : BOOL;
    xStop  : BOOL;
END_VAR
VAR_OUTPUT
    rLastUs : REAL;             // 最近一次段耗时 µs
    rAvgUs  : REAL;
    rMaxUs  : REAL;
    nSamples: DINT;
END_VAR
VAR
    tT0     : LTIME;
    xArmed  : BOOL;
    rSumUs  : LREAL;
END_VAR

IF xStart THEN
    tT0 := LTIME();             // CODESYS 3.5 高精度单调时钟(ns 分辨率)
    xArmed := TRUE;
END_IF
IF xStop AND xArmed THEN
    rLastUs := LREAL_TO_REAL(LTIME_TO_LREAL(LTIME() - tT0) / 1000.0);   // ns→µs
    rSumUs := rSumUs + rLastUs;
    nSamples := nSamples + 1;
    IF rLastUs > rMaxUs THEN rMaxUs := rLastUs; END_IF
    rAvgUs := LREAL_TO_REAL(rSumUs / DINT_TO_LREAL(nSamples));
    xArmed := FALSE;
END_IF
END_FUNCTION_BLOCK

(* ---------- FB_BuildVisuPath:生成 L 形路径点(决赛可视化路径展示) ----------
   物理走线按"先水平后垂直"展开为逐格路径点(曼哈顿口径);
   执行时间按切比雪夫另算 —— 两口径并列,呼应 C2。 *)
FUNCTION_BLOCK FB_BuildVisuPath
VAR_INPUT
    xExecute : BOOL;
    iToX     : INT;
    iToY     : INT;
END_VAR
VAR_OUTPUT
    xDone : BOOL;
END_VAR
VAR
    xOld : BOOL;
    n, x, y : INT;
END_VAR

IF xExecute AND NOT xOld THEN
    n := 0;
    IF iToX >= 0 AND iToX <= GVL_Param.COLS - 1 AND iToY >= 0 AND iToY <= GVL_Param.TIERS - 1 THEN
        FOR x := 0 TO iToX DO                       // 水平段(含起点(0,0))
            GVL_Visu.VisuPathX[n] := x;  GVL_Visu.VisuPathY[n] := 0;  n := n + 1;
        END_FOR
        FOR y := 1 TO iToY DO                       // 垂直段
            GVL_Visu.VisuPathX[n] := iToX;  GVL_Visu.VisuPathY[n] := y;  n := n + 1;
        END_FOR
        GVL_Visu.VisuTargetX := iToX;  GVL_Visu.VisuTargetY := iToY;
        GVL_Visu.VisuPathLen  := FC_CalcPathLen(x0 := 0, y0 := 0, x1 := iToX, y1 := iToY);
        GVL_Visu.VisuExecTime := FC_CalcTravelTime(x0 := 0, y0 := 0, x1 := iToX, y1 := iToY,
                                                   xSimXY := GVL_Param.xSimultaneousXY);
    END_IF
    GVL_Visu.VisuPathCount := n;
    xDone := TRUE;
END_IF
xOld := xExecute;
END_FUNCTION_BLOCK

(* ---------- FB_VisuRefresh:可视化镜像刷新(L6,PRG_Main 尾部每周期常驻调用) ----------
   职责=把"算法语义层"翻译成"画面显示层",三件事:
   1. VisuSlotState[列,层] → VisuSlotColor[列,显示行]:状态→颜色查表 + 上下翻转
      (仓库层0在底、画面行0在顶,显示行 = TIERS-1-层)——画面矩形阵列只绑颜色数组;
   2. 路径叠加:VisuPath 各点在颜色层画蓝,但只叠加在空闲/预占格上
      (不写 VisuSlotState 语义层,避免"蓝色盖掉已占格后无法恢复"的状态污染);
   3. 堆垛机像素坐标:VisuCurrentX/Y(格)→ VisuCraneXpx/Ypx(px,含翻转),
      供堆垛机图元的 Absolute movement 绑定(图元设计位置放 (0,0),偏移即绝对)。
   开销:400 次查表+少量换算/周期 ≈ 微秒级,常驻无压力(L4 实测口径可佐证)。 *)
FUNCTION_BLOCK FB_VisuRefresh
VAR
    c, rw, k, iSt : INT;   // rw=显示行(r/s 是 IEC 置复位保留字,不可作变量名——0706 无头编译揪出的潜伏 bug)
    iT       : INT;        // 设计坐标层(=TIERS-1-rw)
    rHeatMax : REAL;       // C2 频次热力归一分母
    nOpsMax  : INT;        // C6 履历热力归一分母
END_VAR

// 0) C2/C6 热力归一分母(每周期 400 扫;量级远低于既有双重渲染循环)
IF GVL_Visu.iViewMode = 1 THEN
    rHeatMax := 0.0;
    FOR c := 0 TO GVL_Param.COLS - 1 DO
        FOR iT := 0 TO GVL_Param.TIERS - 1 DO
            IF GVL_WH.aSlotFreq[c, iT] > rHeatMax THEN rHeatMax := GVL_WH.aSlotFreq[c, iT]; END_IF
        END_FOR
    END_FOR
ELSIF GVL_Visu.iViewMode = 2 THEN
    nOpsMax := 0;
    FOR c := 0 TO GVL_Param.COLS - 1 DO
        FOR iT := 0 TO GVL_Param.TIERS - 1 DO
            IF GVL_WH.aSlotOps[c, iT] > nOpsMax THEN nOpsMax := GVL_WH.aSlotOps[c, iT]; END_IF
        END_FOR
    END_FOR
END_IF

// 1) 色源三视图 + 上下翻转(显示行 rw=0 是画面顶=层19)
//    优先级:快照对比(CmdCompareMode)> 热力视图(iViewMode 1/2)> 状态视图;
//    热力视图=分析视图:有货格按热力色阶,无货格降级灰系(推荐黄/路径蓝不叠,
//    检修紫仍由 2b 恒显);色表仍 FC_StateToColor/FC_HeatColor 单源。
FOR c := 0 TO GVL_Param.COLS - 1 DO
    FOR rw := 0 TO GVL_Param.TIERS - 1 DO
        iT := GVL_Param.TIERS - 1 - rw;
        IF GVL_Visu.CmdCompareMode AND GVL_Visu.xSnapValid THEN
            GVL_Visu.VisuSlotColor[c, rw] :=
                FC_StateToColor(iState := GVL_Visu.aSnapState[c, iT]);
        ELSIF GVL_Visu.iViewMode = 1 THEN            // C2 频次热力
            IF GVL_WH.aSlots[c, iT].GoodsId > 0 THEN
                GVL_Visu.VisuSlotColor[c, rw] :=
                    FC_HeatColor(rVal := GVL_WH.aSlotFreq[c, iT], rMax := rHeatMax);
            ELSIF GVL_WH.aSlots[c, iT].PresetOcc THEN
                GVL_Visu.VisuSlotColor[c, rw] := FC_StateToColor(iState := 1);
            ELSE
                GVL_Visu.VisuSlotColor[c, rw] := FC_StateToColor(iState := 0);
            END_IF
        ELSIF GVL_Visu.iViewMode = 2 THEN            // C6 损耗履历热力
            IF GVL_WH.aSlotOps[c, iT] > 0 THEN
                GVL_Visu.VisuSlotColor[c, rw] :=
                    FC_HeatColor(rVal := INT_TO_REAL(GVL_WH.aSlotOps[c, iT]),
                                 rMax := INT_TO_REAL(nOpsMax));
            ELSIF GVL_WH.aSlots[c, iT].PresetOcc THEN
                GVL_Visu.VisuSlotColor[c, rw] := FC_StateToColor(iState := 1);
            ELSE
                GVL_Visu.VisuSlotColor[c, rw] := FC_StateToColor(iState := 0);
            END_IF
        ELSE                                          // 状态视图(原逻辑)
            GVL_Visu.VisuSlotColor[c, rw] :=
                FC_StateToColor(iState := GVL_Visu.VisuSlotState[c, iT]);
        END_IF
    END_FOR
END_FOR

// 2) 路径叠加(蓝):仅状态视图;只画在空闲/预占格上;对比模式跳过(快照是纯布局对比)
IF GVL_Visu.iViewMode = 0
   AND NOT (GVL_Visu.CmdCompareMode AND GVL_Visu.xSnapValid) THEN
    FOR k := 0 TO GVL_Visu.VisuPathCount - 1 DO
        IF k > 39 THEN EXIT; END_IF                   // 路径数组上限 40 点,防越界
        iSt := GVL_Visu.VisuSlotState[GVL_Visu.VisuPathX[k], GVL_Visu.VisuPathY[k]];
        IF iSt = 0 OR iSt = 1 THEN
            GVL_Visu.VisuSlotColor[GVL_Visu.VisuPathX[k],
                                   GVL_Param.TIERS - 1 - GVL_Visu.VisuPathY[k]] :=
                FC_StateToColor(iState := 4);
        END_IF
    END_FOR
END_IF

// 2b) A3 检修叠加(恒显:物理状态,独立于布局/快照/路径/热力;Reset 不清)
FOR c := 0 TO GVL_Param.COLS - 1 DO
    FOR rw := 0 TO GVL_Param.TIERS - 1 DO
        IF GVL_WH.aMaintBlock[c, GVL_Param.TIERS - 1 - rw] THEN
            GVL_Visu.VisuSlotColor[c, rw] := FC_StateToColor(iState := 7);
        END_IF
    END_FOR
END_FOR

// 2c) C1 层高亮(选中层整行向白混色 45%,叠在一切色源之上;顺带数该层在货格)
GVL_Visu.VisuTierOcc := 0;
IF GVL_Visu.InTierSel >= 0 AND GVL_Visu.InTierSel <= GVL_Param.TIERS - 1 THEN
    rw := GVL_Param.TIERS - 1 - GVL_Visu.InTierSel;
    FOR c := 0 TO GVL_Param.COLS - 1 DO
        GVL_Visu.VisuSlotColor[c, rw] := FC_BlendLight(dw := GVL_Visu.VisuSlotColor[c, rw]);
        IF GVL_WH.aSlots[c, GVL_Visu.InTierSel].GoodsId > 0 THEN
            GVL_Visu.VisuTierOcc := GVL_Visu.VisuTierOcc + 1;
        END_IF
    END_FOR
END_IF

// 3) 堆垛机格坐标 → 像素坐标(图元锚点=左上角,大小=一个单元格)
GVL_Visu.VisuCraneXpx := GVL_Param.GRID_X0 + GVL_Visu.VisuCurrentX * GVL_Param.CELL_PX_W;
GVL_Visu.VisuCraneYpx := GVL_Param.GRID_Y0
    + (GVL_Param.TIERS - 1 - GVL_Visu.VisuCurrentY) * GVL_Param.CELL_PX_H;
END_FUNCTION_BLOCK

(* ---------- FB_GoodsInput:交互货物输入封装(评分细则6/7;0707 T2.2 从 PRG_Main 抽取) ----------
   功能:题面五属性(序号/名称/重量/频次/体积)输入 → 边界校验 → 写入货物表 → 即时推荐仓位。
         把"关键交互算法封装为功能块,IO 参数设计合理"(评分细则6)显式化。
   输入:xAdd 上升沿触发;iId/sName/rWeight/rFreq/rVolume = 题面五属性。
   输出:xOk 成功入表;xFound 有推荐位;iSugX/iSugY 推荐列/层;
         iErrId 错误码 0=ok / 1=满仓 / 2=负输入 / 3=无可行位。
   边界:满仓(≥MAX_GOODS)→iErrId=1;任一属性<0→iErrId=2;无可行位(如超重货)→iErrId=3。
   示例:xAdd 上升沿+合法轻货 → xOk=TRUE,xFound=TRUE,iSug=近位;超重货 → xOk=TRUE,iErrId=3。
   分层:可视化(推荐高亮/路径叠加/状态文本/报警灯)由调用方 PRG_Main 按本 FB 输出编排——
         本 FB 只算(可单元测试),PRG_Main 只画(画面职责)。 *)
FUNCTION_BLOCK FB_GoodsInput
VAR_INPUT
    xAdd    : BOOL;             // 添加触发(上升沿)
    iId     : INT;
    sName   : STRING[32];
    rWeight : REAL;
    rFreq   : REAL;
    rVolume : REAL;
END_VAR
VAR_OUTPUT
    xOk     : BOOL;             // 本次是否成功入表
    xFound  : BOOL;             // 是否有推荐仓位
    iSugX   : INT;              // 推荐列
    iSugY   : INT;              // 推荐层
    iErrId  : INT;             // 0=ok 1=满仓 2=负输入 3=无可行位
END_VAR
VAR
    xOld    : BOOL;
    i       : INT;
    rWMaxTmp, rFMaxTmp : REAL;
    fbSel   : FB_SelectSlot;
END_VAR

xOk := FALSE;  xFound := FALSE;  iErrId := 0;  iSugX := -1;  iSugY := -1;
IF xAdd AND NOT xOld THEN
    IF GVL_WH.iGoodsCount >= GVL_Param.MAX_GOODS THEN
        iErrId := 1;                                    // 边界:满仓拒收
    ELSIF rWeight < 0.0 OR rFreq < 0.0 OR rVolume < 0.0 THEN
        iErrId := 2;                                    // 边界:负属性拒收
    ELSE
        GVL_WH.iGoodsCount := GVL_WH.iGoodsCount + 1;
        GVL_WH.aGoods[GVL_WH.iGoodsCount].Id       := iId;
        GVL_WH.aGoods[GVL_WH.iGoodsCount].Name     := sName;
        GVL_WH.aGoods[GVL_WH.iGoodsCount].Weight   := rWeight;
        GVL_WH.aGoods[GVL_WH.iGoodsCount].Freq     := rFreq;
        GVL_WH.aGoods[GVL_WH.iGoodsCount].Volume   := rVolume;
        GVL_WH.aGoods[GVL_WH.iGoodsCount].Assigned := FALSE;
        xOk := TRUE;
        // 即时推荐(归一分母取当前批次最大,与 score 口径一致)
        rWMaxTmp := MAX(rWeight, 1.0);  rFMaxTmp := MAX(rFreq, 1.0);
        FOR i := 1 TO GVL_WH.iGoodsCount DO
            IF GVL_WH.aGoods[i].Weight > rWMaxTmp THEN rWMaxTmp := GVL_WH.aGoods[i].Weight; END_IF
            IF GVL_WH.aGoods[i].Freq   > rFMaxTmp THEN rFMaxTmp := GVL_WH.aGoods[i].Freq;   END_IF
        END_FOR
        fbSel(iStrategy := 2, rGoodW := rWeight, rGoodF := rFreq, rGoodV := rVolume,
              rWMax := rWMaxTmp, rFMax := rFMaxTmp);
        IF fbSel.xFound THEN
            xFound := TRUE;  iSugX := fbSel.iBestX;  iSugY := fbSel.iBestY;
        ELSE
            iErrId := 3;                                // 无可行位(如超重货连底层都放不下)
        END_IF
    END_IF
END_IF
xOld := xAdd;
END_FUNCTION_BLOCK

(* ---------- FB_QueryGood:单件查询(评分细则8"统计信息";块3 P3 查询页) ----------
   功能:按序号扫货物表 → 五属性+位置+路径长/行程时间(存量口径)+载货行程/装卸档
        (U2 拟真对照,调参区改 rLadenFactorVY/装卸三档此二值实时变)→ 网格青色高亮。
   输入:xQuery 上升沿触发;iId 查询序号。
   输出:直接写 GVL_Visu.Qry* 组(画面服务 FB,同 FB_VisuRefresh 先例);
        高亮=VisuSlotState 置 6,旧高亮恢复为 2(命中货必 Assigned=原状态已占用)。
   边界:iId<=0 → QryFound=FALSE;未找到 → 全字段清零;未分配货 → 位置=-1、时间组=0。
   示例:查演示批 Id=1 → QryFound=TRUE,位置/时间齐,该格变青;查 Id=999 → FALSE。 *)
FUNCTION_BLOCK FB_QueryGood
VAR_INPUT
    xQuery : BOOL;              // 查询触发(上升沿)
    iId    : INT;               // 查询序号
END_VAR
VAR
    xOld   : BOOL;
    i      : INT;
    iLastX : INT := -1;         // 上次高亮列(-1=无,清除用)
    iLastY : INT := -1;         // 上次高亮层
END_VAR

IF xQuery AND NOT xOld THEN
    // 清上次青色高亮(只清仍=6 的格,防误清其他状态;恢复为 2=已占用)
    IF iLastX >= 0 AND iLastY >= 0 THEN
        IF GVL_Visu.VisuSlotState[iLastX, iLastY] = 6 THEN
            GVL_Visu.VisuSlotState[iLastX, iLastY] := 2;
        END_IF
        iLastX := -1;  iLastY := -1;
    END_IF
    // 输出组清零(未命中时字段不残留上次结果)
    GVL_Visu.QryFound := FALSE;
    GVL_Visu.QryX := -1;            GVL_Visu.QryY := -1;
    GVL_Visu.QryName := '';         GVL_Visu.QryWeight := 0.0;
    GVL_Visu.QryFreq := 0.0;        GVL_Visu.QryVolume := 0.0;
    GVL_Visu.QryPathLen := 0.0;     GVL_Visu.QryExecTime := 0.0;
    GVL_Visu.QryTravelLaden := 0.0; GVL_Visu.QryHandleT := 0.0;
    IF iId > 0 THEN                                   // 边界:非正序号直接未找到
        FOR i := 1 TO GVL_WH.iGoodsCount DO
            IF GVL_WH.aGoods[i].Id = iId THEN
                GVL_Visu.QryFound  := TRUE;
                GVL_Visu.QryName   := GVL_WH.aGoods[i].Name;
                GVL_Visu.QryWeight := GVL_WH.aGoods[i].Weight;
                GVL_Visu.QryFreq   := GVL_WH.aGoods[i].Freq;
                GVL_Visu.QryVolume := GVL_WH.aGoods[i].Volume;
                IF GVL_WH.aGoods[i].Assigned THEN
                    GVL_Visu.QryX        := GVL_WH.aGoods[i].X;
                    GVL_Visu.QryY        := GVL_WH.aGoods[i].Y;
                    GVL_Visu.QryPathLen  := GVL_WH.aGoods[i].PathLength;
                    GVL_Visu.QryExecTime := GVL_WH.aGoods[i].ExecTime;
                    // U2 拟真对照:载货行程(垂直折减)+ 装卸三档(调参区实时联动)
                    GVL_Visu.QryTravelLaden := FC_TravelLaden(
                        x0 := 0, y0 := 0,
                        x1 := GVL_WH.aGoods[i].X, y1 := GVL_WH.aGoods[i].Y,
                        xSimXY := GVL_Param.xSimultaneousXY);
                    GVL_Visu.QryHandleT := FC_HandleTime(rW := GVL_WH.aGoods[i].Weight);
                    // 青色高亮 + 记住位置供下次清除
                    GVL_Visu.VisuSlotState[GVL_WH.aGoods[i].X, GVL_WH.aGoods[i].Y] := 6;
                    iLastX := GVL_WH.aGoods[i].X;
                    iLastY := GVL_WH.aGoods[i].Y;
                END_IF
                EXIT;                                 // 序号唯一,命中即止
            END_IF
        END_FOR
    END_IF
END_IF
xOld := xQuery;
END_FUNCTION_BLOCK

(* ---------- FB_RecordPage:统计记录页 10 行窗口(评分细则8;块3 P2) ----------
   功能:aGoods 全表 → 10 行显示窗口(aRow* 并行数组),翻页上升沿±10 并钳位;
        每周期常驻刷新(数据总最新;40 次数组访问,微秒级)。
   设计:窗口映射而非 400 行整表 —— WebVisu 渲染预算(画面标准 §6)+ 一屏一焦点(§3)。
   输入:xPageUp/xPageDown 翻页按钮(上升沿)。
   输出:直接写 GVL_Visu.aRow*/iRecTop/iRecTotal(画面服务 FB)。
   边界:iRecTop 钳位 [1, max(1, iGoodsCount-9)];窗口越界行 Id=0(画面按 0 显示空行);
        未分配货位置=-1、数值=0(与查询页口径一致)。
   示例:120 件表,iRecTop=1 显示 1..10;PageDown→11..20;拉到底 111..120 后再按不动。 *)
FUNCTION_BLOCK FB_RecordPage
VAR_INPUT
    xPageUp   : BOOL;           // 上翻(上升沿,-10)
    xPageDown : BOOL;           // 下翻(上升沿,+10)
END_VAR
VAR
    xUpOld, xDnOld : BOOL;
    k, idx         : INT;
END_VAR

// 翻页(上升沿)
IF xPageUp AND NOT xUpOld THEN
    GVL_Visu.iRecTop := GVL_Visu.iRecTop - 10;
END_IF
IF xPageDown AND NOT xDnOld THEN
    GVL_Visu.iRecTop := GVL_Visu.iRecTop + 10;
END_IF
xUpOld := xPageUp;
xDnOld := xPageDown;

// 钳位:上限先于下限(空表时两界都收敛到 1)
IF GVL_Visu.iRecTop > GVL_WH.iGoodsCount - 9 THEN
    GVL_Visu.iRecTop := GVL_WH.iGoodsCount - 9;
END_IF
IF GVL_Visu.iRecTop < 1 THEN
    GVL_Visu.iRecTop := 1;
END_IF
GVL_Visu.iRecTotal := GVL_WH.iGoodsCount;

// 10 行窗口映射(常驻:批量分配进行中翻表也能看到最新位置)
FOR k := 0 TO 9 DO
    idx := GVL_Visu.iRecTop + k;
    IF idx >= 1 AND idx <= GVL_WH.iGoodsCount THEN
        GVL_Visu.aRowId[k] := GVL_WH.aGoods[idx].Id;
        IF GVL_WH.aGoods[idx].Assigned THEN
            GVL_Visu.aRowX[k]       := GVL_WH.aGoods[idx].X;
            GVL_Visu.aRowY[k]       := GVL_WH.aGoods[idx].Y;
            GVL_Visu.aRowPathLen[k] := GVL_WH.aGoods[idx].PathLength;
            GVL_Visu.aRowExecT[k]   := GVL_WH.aGoods[idx].ExecTime;
        ELSE
            GVL_Visu.aRowX[k]       := -1;    // 未分配:位置=-1(画面显示 "-")
            GVL_Visu.aRowY[k]       := -1;
            GVL_Visu.aRowPathLen[k] := 0.0;
            GVL_Visu.aRowExecT[k]   := 0.0;
        END_IF
    ELSE
        GVL_Visu.aRowId[k]      := 0;         // 越界:空行(Id=0 约定)
        GVL_Visu.aRowX[k]       := -1;
        GVL_Visu.aRowY[k]       := -1;
        GVL_Visu.aRowPathLen[k] := 0.0;
        GVL_Visu.aRowExecT[k]   := 0.0;
    END_IF
END_FOR
END_FUNCTION_BLOCK

(* ---------- FB_SceneDetect:场景检测器(A2 驾驶舱连击,0711) ----------
   sim/strategy_lib.py 的 batch_profile + select_strategy(holistic 档)忠实 ST 化:
   批次画像(n/density/skew/w_mean/w_heavy)一次遍历+分片排序算出,阈值级联推荐策略。
   档位说明:holistic=题面全要素默认档(重货低层 C6/能耗 C4 权重高,AWRA 主推,
   极小批+无画像信息降级简单规则=F18-2);lex/speed 档推荐 TOB/CB,PLC 策略库未含
   (sim 层 A1 实验已证 lex 档达 oracle 98.5%),ST 版按主打叙事实现 holistic 档。
   skew=top20% 件频次占比:需频次降序排序——插入排序按件分片(每周期 nPerCycle 件,
   单件插入最坏 O(n) 步,n=400 时单周期约 2 万步 REAL 比较,远低于分片先例
   nPairsPerCycle=200 对评分的量级,不触发看门狗)。
   触发:iGoodsCount 变化自动重算(演示:载批/加件即刷新);xForce 强制重算
   (货物属性原地变更时用,如测试)。运行中数据再变=丢弃重来(以终值为准)。
   输出推荐档位用 SelStrategy 语义:1=near(COL) 2=score 3=AWRA-LS。 *)
FUNCTION_BLOCK FB_SceneDetect
VAR_INPUT
    xForce      : BOOL;             // 上升沿:强制重算(iGoodsCount 未变但属性变了)
END_VAR
VAR_OUTPUT
    xValid      : BOOL;             // 画像+推荐已就绪(n=0 时 FALSE)
    iRecBatch   : INT := -1;        // 批量模式推荐(整批画像已知,演示主口径)
    iRecOnline  : INT := -1;        // 在线模式推荐(逐件到货口径,F18-2)
END_VAR
VAR
    iStep       : INT := 0;         // 0=空闲 1=排序分片中 2=完成
    iCntLast    : INT := -1;        // 上次看到的货物数(变化检测)
    xForceOld   : BOOL;
    aF          : ARRAY[1..400] OF REAL;    // 频次工作数组(降序)
    iSorted     : INT;              // 已插入排序的件数
    nPerCycle   : INT := 50;        // 每周期插入件数(分片粒度)
    i, j, iTop  : INT;
    rV, rSumAll, rSumTop, rWSum : REAL;
    iHeavy, nLoc : INT;
    rSkew       : REAL;
END_VAR

// 触发检测:货物数变化 或 强制重算 → 从头开始
IF (GVL_WH.iGoodsCount <> iCntLast) OR (xForce AND NOT xForceOld) THEN
    iCntLast := GVL_WH.iGoodsCount;
    IF GVL_WH.iGoodsCount = 0 THEN
        xValid := FALSE;  iStep := 0;
        iRecBatch := -1;  iRecOnline := -1;
        GVL_Visu.VisuProfN := 0;        GVL_Visu.VisuProfDensity := 0.0;
        GVL_Visu.VisuProfSkew := 0.0;   GVL_Visu.VisuProfWMean := 0.0;
        GVL_Visu.VisuProfWHeavy := 0.0; GVL_Visu.VisuRecStrategy := -1;
        GVL_Visu.VisuRecText := 'DET_NO_DATA';
    ELSE
        xValid := FALSE;  iStep := 1;  iSorted := 0;
        rWSum := 0.0;  iHeavy := 0;  rSumAll := 0.0;
        // 一次遍历:重量均值/重货占比/频次总和(排序前先取齐标量特征)
        FOR i := 1 TO GVL_WH.iGoodsCount DO
            aF[i] := GVL_WH.aGoods[i].Freq;
            rSumAll := rSumAll + aF[i];
            rWSum := rWSum + GVL_WH.aGoods[i].Weight;
            IF GVL_WH.aGoods[i].Weight > 60.0 THEN iHeavy := iHeavy + 1; END_IF
        END_FOR
    END_IF
END_IF
xForceOld := xForce;

// 分片排序:每周期把 nPerCycle 件插入已排序前缀(降序,稳定=Python sorted 语义)
IF iStep = 1 THEN
    nLoc := GVL_WH.iGoodsCount;
    j := iSorted + 1;
    WHILE (j <= nLoc) AND (j <= iSorted + nPerCycle) DO
        rV := aF[j];
        i := j - 1;
        WHILE i >= 1 DO                      // IEC AND 不短路:下标判断与访问分离防 aF[0] 越界
            IF aF[i] < rV THEN               // 严格小于才后移=稳定排序(同值保原序)
                aF[i + 1] := aF[i];
                i := i - 1;
            ELSE
                EXIT;
            END_IF
        END_WHILE
        aF[i + 1] := rV;
        j := j + 1;
    END_WHILE
    iSorted := j - 1;
    IF iSorted >= nLoc THEN
        // ---- 完成拍:算画像 + 阈值级联推荐(与 strategy_lib v1 同逻辑) ----
        iTop := MAX(1, nLoc / 5);
        rSumTop := 0.0;
        FOR i := 1 TO iTop DO rSumTop := rSumTop + aF[i]; END_FOR
        IF rSumAll > 0.0 THEN rSkew := rSumTop / rSumAll; ELSE rSkew := 0.0; END_IF
        GVL_Visu.VisuProfN       := nLoc;
        GVL_Visu.VisuProfDensity := INT_TO_REAL(nLoc) / 267.0;   // sum 口径可用位
        GVL_Visu.VisuProfSkew    := rSkew;
        GVL_Visu.VisuProfWMean   := rWSum / INT_TO_REAL(nLoc);
        GVL_Visu.VisuProfWHeavy  := INT_TO_REAL(iHeavy) / INT_TO_REAL(nLoc);
        // holistic 批量档:极小批+无画像→near,否则 AWRA(全要素安全档)
        IF rSkew < 0.35 AND nLoc <= 20 THEN
            iRecBatch := 1;
            GVL_Visu.VisuRecText := 'REC=NEAR_TINY_FLAT';
        ELSE
            iRecBatch := 3;
            GVL_Visu.VisuRecText := 'REC=AWRA_HOLISTIC';
        END_IF
        // 在线档(F18-2):画像无信息量 或 极小批→near,否则 score
        IF rSkew < 0.35 OR nLoc <= 20 THEN
            iRecOnline := 1;
        ELSE
            iRecOnline := 2;
        END_IF
        GVL_Visu.VisuRecStrategy := iRecBatch;
        xValid := TRUE;
        iStep := 2;
    END_IF
END_IF
END_FUNCTION_BLOCK

(* ---------- FB_UserAuth:两级权限登录(A4 变量层,0711) ----------
   方案依据(0711 官方文档核实):内置 visu Access Rights 只能 IDE 逐元素手工配、
   无 ScriptEngine 接口,与画面生成管线不兼容→变量层;画面元素锁定(Deactivated/
   Invisible 绑 iUserLevel<1)+ FB_ParamGuard 回滚构成双闸。
   已知坑对策:①PIN 消费即清(PRG_Main 登录后清 InPinCode,画面无回显元件);
   ②iLevel 非 RETAIN(断电回操作员=安全默认);③单客户端演示口径,多客户端需
   CurrentClientId 隔离(报告局限性章如实写)。演示 PIN=GVL_Param.ADMIN_PIN,非真实凭据。 *)
FUNCTION_BLOCK FB_UserAuth
VAR_INPUT
    xLogin  : BOOL;                 // 上升沿:按当前 iPin 尝试登录
    iPin    : INT;
    xLogout : BOOL;                 // 上升沿:登出回操作员
END_VAR
VAR_OUTPUT
    iLevel    : INT := 0;           // 0=操作员 1=管理员
    sUserText : STRING[32] := 'USER=OPERATOR';
    iFailCnt  : INT := 0;           // 失败计数(演示可见,防猜码叙事)
END_VAR
VAR
    xLoginOld, xLogoutOld : BOOL;
END_VAR

IF xLogin AND NOT xLoginOld THEN
    IF iPin = GVL_Param.ADMIN_PIN THEN
        iLevel := 1;
        sUserText := 'USER=ADMIN';
    ELSE
        iFailCnt := iFailCnt + 1;
        sUserText := 'LOGIN_FAIL';
    END_IF
END_IF
IF xLogout AND NOT xLogoutOld THEN
    iLevel := 0;
    sUserText := 'USER=OPERATOR';
END_IF
xLoginOld := xLogin;
xLogoutOld := xLogout;
END_FUNCTION_BLOCK

(* ---------- FB_ParamGuard:调参守卫(A4 双闸之二,0711) ----------
   变量层权限的 ST 侧闸门:管理员在位时实时快照全部可调参数;操作员级时每周期
   把参数回滚到快照——即使画面元素锁定被绕过(如元素漏绑权限表达式),
   非管理员的改动存活不超过一个扫描周期。守卫集=GVL_Param 变量段全部可调项;
   SelStrategy/xAutoStrategy/检修命令不在守卫集(操作员演示职能,检修另有权限门)。 *)
FUNCTION_BLOCK FB_ParamGuard
VAR_INPUT
    iLevel : INT;                   // 当前用户级(FB_UserAuth.iLevel)
END_VAR
VAR
    xInit : BOOL := TRUE;           // 首周期:快照=现值(防 FB 初值 0 反灌参数)
    sVx, sVy, sTLoad, sTUnload, sAx, sAy          : REAL;
    sLadenVY, sHW1, sHW2, sHT1, sHT2, sHT3        : REAL;
    sAlpha, sBeta, sGamma, sDelta, sL1, sL2, sL3  : REAL;
    sSimXY, sUseAccel                             : BOOL;
    sPreRule, sBatchPC, sPairsPC, sMaxLsR         : INT;
END_VAR

IF xInit OR iLevel >= 1 THEN
    // 管理员在位(或首周期):放行并持续刷新快照——管理员改的值即新基准
    sVx := GVL_Param.rVx;                  sVy := GVL_Param.rVy;
    sTLoad := GVL_Param.rTLoad;            sTUnload := GVL_Param.rTUnload;
    sAx := GVL_Param.rAx;                  sAy := GVL_Param.rAy;
    sLadenVY := GVL_Param.rLadenFactorVY;
    sHW1 := GVL_Param.rHandleW1;           sHW2 := GVL_Param.rHandleW2;
    sHT1 := GVL_Param.rHandleT1;           sHT2 := GVL_Param.rHandleT2;
    sHT3 := GVL_Param.rHandleT3;
    sAlpha := GVL_Param.rAlpha;            sBeta := GVL_Param.rBeta;
    sGamma := GVL_Param.rGamma;            sDelta := GVL_Param.rDelta;
    sL1 := GVL_Param.rLambda1;             sL2 := GVL_Param.rLambda2;
    sL3 := GVL_Param.rLambda3;
    sSimXY := GVL_Param.xSimultaneousXY;   sUseAccel := GVL_Param.xUseAccel;
    sPreRule := GVL_Param.iPreRule;        sBatchPC := GVL_Param.nBatchPerCycle;
    sPairsPC := GVL_Param.nPairsPerCycle;  sMaxLsR := GVL_Param.nMaxLsRounds;
    xInit := FALSE;
ELSE
    // 操作员级:任何参数偏离快照即回滚(下周期生效,画面可见值跳回)
    GVL_Param.rVx := sVx;                  GVL_Param.rVy := sVy;
    GVL_Param.rTLoad := sTLoad;            GVL_Param.rTUnload := sTUnload;
    GVL_Param.rAx := sAx;                  GVL_Param.rAy := sAy;
    GVL_Param.rLadenFactorVY := sLadenVY;
    GVL_Param.rHandleW1 := sHW1;           GVL_Param.rHandleW2 := sHW2;
    GVL_Param.rHandleT1 := sHT1;           GVL_Param.rHandleT2 := sHT2;
    GVL_Param.rHandleT3 := sHT3;
    GVL_Param.rAlpha := sAlpha;            GVL_Param.rBeta := sBeta;
    GVL_Param.rGamma := sGamma;            GVL_Param.rDelta := sDelta;
    GVL_Param.rLambda1 := sL1;             GVL_Param.rLambda2 := sL2;
    GVL_Param.rLambda3 := sL3;
    GVL_Param.xSimultaneousXY := sSimXY;   GVL_Param.xUseAccel := sUseAccel;
    GVL_Param.iPreRule := sPreRule;        GVL_Param.nBatchPerCycle := sBatchPC;
    GVL_Param.nPairsPerCycle := sPairsPC;  GVL_Param.nMaxLsRounds := sMaxLsR;
END_IF
END_FUNCTION_BLOCK

(* ---- 09_FB_ScanLoadProbeNs_备用.st ---- *)
(* ============================================================
   09_FB_ScanLoadProbeNs_备用.st — L4 兜底探针(候选③:SysTime 库时钟源)
   ⚠️ 备用件:仅当信箱批次 0705-B 的任务监视页读数也恒为 0 时才导入,平时不进工程。

   为什么要有它(root cause 记录):
   FB_ScanLoadProbe 用 LTIME() 差分,在 AB 仿真中恒为 0。最可能根因不是"分辨率不够",
   而是 **IEC 时间函数在一个扫描周期内返回缓存值**(任务开始时取一次,周期内不变)——
   若如此,"累计窗口摊薄法"(原候选②)同样无效:窗口内累加的每段差分仍是 0。
   兜底必须换时钟源:SysTime 库的 SysTimeGetNs/SysTimeGetUs 直接调操作系统计时器,
   不走 IEC 周期缓存。故候选顺序修订为 ①任务监视页 → ③本文件 → ④真机。

   导入方法(仅在需要时):
   1. AB 里 Application 下 Library Manager(库管理器)→ Add Library(添加库)→
      搜索 "SysTime"(SysTime, System 分类)→ 添加。找不到该库 → 停,截图汇报。
   2. 添加 POU-功能块 FB_ScanLoadProbeNs,粘贴本文件下方代码。
   3. 编译若报 SysTimeGetNs 参数名不符:在实现区把 SysTimeGetNs( 重新输入,
      按 AB 输入助手(F2)提示的形参名改(不同版本形参名可能是 pTimeNs/pUsTime 等,
      功能相同:把当前纳秒计数写进传入变量)。改完把实际形参名写进汇报。
   4. PLC_PRG 接线与原探针完全相同(fbProbeNs 换名即可),接口刻意保持一致。
   ============================================================ *)

FUNCTION_BLOCK FB_ScanLoadProbeNs
VAR_INPUT
    xStart : BOOL;              // 段前置 TRUE
    xStop  : BOOL;              // 段后置 TRUE
END_VAR
VAR_OUTPUT
    rLastUs : REAL;             // 最近一次段耗时 µs
    rAvgUs  : REAL;
    rMaxUs  : REAL;
    nSamples: DINT;
END_VAR
VAR
    tT0     : SYSTIME;          // 段前时刻 ns(SYSTIME=ULINT,SysTime 库定义)
    tT1     : SYSTIME;          // 段后时刻 ns
    xArmed  : BOOL;             // 已记录段前时刻,等待段后
    rSumUs  : LREAL;            // 累计和用 LREAL,防长跑精度丢失
    rDiffUs : REAL;
END_VAR

// 段前:取一次系统纳秒计数(直连 OS 计时器,不受 IEC 周期缓存影响)
IF xStart AND NOT xArmed THEN
    SysTimeGetNs(pTimeNs := tT0);   // 形参名以 AB 输入助手为准,见文件头第3条
    xArmed := TRUE;
END_IF

// 段后:再取一次,差分入统计
IF xStop AND xArmed THEN
    SysTimeGetNs(pTimeNs := tT1);
    xArmed := FALSE;
    IF tT1 >= tT0 THEN                               // 防计数器回绕的负差
        rDiffUs := ULINT_TO_REAL(tT1 - tT0) / 1000.0;   // ns → µs
        rLastUs := rDiffUs;
        nSamples := nSamples + 1;
        rSumUs := rSumUs + REAL_TO_LREAL(rDiffUs);
        rAvgUs := LREAL_TO_REAL(rSumUs / DINT_TO_LREAL(nSamples));
        IF rDiffUs > rMaxUs THEN rMaxUs := rDiffUs; END_IF
    END_IF
END_IF
END_FUNCTION_BLOCK
